# B&R Automation Studio project AAU12Segmenter (part 5)

#### linkMovement.st
```iecst
ACTION linkMovementProgram:
	//Setup
	positionContainerLinkMovement[0].Shuttle1.xPos := 0.120;
	positionContainerLinkMovement[0].Shuttle1.yPos := 0.120;
	positionContainerLinkMovement[0].Shuttle2.xPos := 0.360;
	positionContainerLinkMovement[0].Shuttle2.yPos := 0.360;
	positionContainerLinkMovement[0].Shuttle3.xPos := 0.360;
	positionContainerLinkMovement[0].Shuttle3.yPos := 0.120;
	positionContainerLinkMovement[0].Shuttle4.xPos := 0.120;
	positionContainerLinkMovement[0].Shuttle4.yPos := 0.360;

	positionContainerLinkMovement[1].Shuttle1.xPos := 0.060;
	positionContainerLinkMovement[1].Shuttle1.yPos := 0.060;
	positionContainerLinkMovement[1].Shuttle2.xPos := 0.180;
	positionContainerLinkMovement[1].Shuttle2.yPos := 0.180;
	positionContainerLinkMovement[1].Shuttle3.xPos := 0.180;
	positionContainerLinkMovement[1].Shuttle3.yPos := 0.060;
	positionContainerLinkMovement[1].Shuttle4.xPos := 0.060;
	positionContainerLinkMovement[1].Shuttle4.yPos := 0.180;

	positionContainerLinkMovement[2].Shuttle1.xPos := 0.120;
	positionContainerLinkMovement[2].Shuttle1.yPos := 0.120;
	positionContainerLinkMovement[2].Shuttle2.xPos := 0.360;
	positionContainerLinkMovement[2].Shuttle2.yPos := 0.360;
	positionContainerLinkMovement[2].Shuttle3.xPos := 0.360;
	positionContainerLinkMovement[2].Shuttle3.yPos := 0.120;
	positionContainerLinkMovement[2].Shuttle4.xPos := 0.120;
	positionContainerLinkMovement[2].Shuttle4.yPos := 0.360;

	positionContainerLinkMovement[3].Shuttle1.xPos := 0.300;
	positionContainerLinkMovement[3].Shuttle1.yPos := 0.060;
	positionContainerLinkMovement[3].Shuttle2.xPos := 0.420;
	positionContainerLinkMovement[3].Shuttle2.yPos := 0.180;
	positionContainerLinkMovement[3].Shuttle3.xPos := 0.420;
	positionContainerLinkMovement[3].Shuttle3.yPos := 0.060;
	positionContainerLinkMovement[3].Shuttle4.xPos := 0.300;
	positionContainerLinkMovement[3].Shuttle4.yPos := 0.180;

	positionContainerLinkMovement[4].Shuttle1.xPos := 0.120;
	positionContainerLinkMovement[4].Shuttle1.yPos := 0.120;
	positionContainerLinkMovement[4].Shuttle2.xPos := 0.360;
	positionContainerLinkMovement[4].Shuttle2.yPos := 0.360;
	positionContainerLinkMovement[4].Shuttle3.xPos := 0.360;
	positionContainerLinkMovement[4].Shuttle3.yPos := 0.120;
	positionContainerLinkMovement[4].Shuttle4.xPos := 0.120;
	positionContainerLinkMovement[4].Shuttle4.yPos := 0.360;

	positionContainerLinkMovement[5].Shuttle1.xPos := 0.300;
	positionContainerLinkMovement[5].Shuttle1.yPos := 0.300;
	positionContainerLinkMovement[5].Shuttle2.xPos := 0.420;
	positionContainerLinkMovement[5].Shuttle2.yPos := 0.420;
	positionContainerLinkMovement[5].Shuttle3.xPos := 0.420;
	positionContainerLinkMovement[5].Shuttle3.yPos := 0.300;
	positionContainerLinkMovement[5].Shuttle4.xPos := 0.300;
	positionContainerLinkMovement[5].Shuttle4.yPos := 0.420;

	positionContainerLinkMovement[6].Shuttle1.xPos := 0.120;
	positionContainerLinkMovement[6].Shuttle1.yPos := 0.120;
	positionContainerLinkMovement[6].Shuttle2.xPos := 0.360;
	positionContainerLinkMovement[6].Shuttle2.yPos := 0.360;
	positionContainerLinkMovement[6].Shuttle3.xPos := 0.360;
	positionContainerLinkMovement[6].Shuttle3.yPos := 0.120;
	positionContainerLinkMovement[6].Shuttle4.xPos := 0.120;
	positionContainerLinkMovement[6].Shuttle4.yPos := 0.360;

	positionContainerLinkMovementNew[0].initXPos := 0.540;
	positionContainerLinkMovementNew[0].initYPos := 0.300;
	positionContainerLinkMovementNew[1].initXPos := 0.540;
	positionContainerLinkMovementNew[1].initYPos := 0.420;
	positionContainerLinkMovementNew[2].initXPos := 0.660;
	positionContainerLinkMovementNew[2].initYPos := 0.540;
	positionContainerLinkMovementNew[3].initXPos := 0.660;
	positionContainerLinkMovementNew[3].initYPos := 0.660;

	positionContainerLinkMovementNew[4].initXPos := 0.120;
	positionContainerLinkMovementNew[4].initYPos := 0.120;
	positionContainerLinkMovementNew[5].initXPos := 0.120;
	positionContainerLinkMovementNew[5].initYPos := 0.240;
	positionContainerLinkMovementNew[6].initXPos := 0.240;
	positionContainerLinkMovementNew[6].initYPos := 0.240;
	positionContainerLinkMovementNew[7].initXPos := 0.240;
	positionContainerLinkMovementNew[7].initYPos := 0.120;
	positionContainerLinkMovementNew[8].initXPos := 0.540;
	positionContainerLinkMovementNew[8].initYPos := 0.900;
	positionContainerLinkMovementNew[9].initXPos := 0.660;
	positionContainerLinkMovementNew[9].initYPos := 0.900;

	CASE em.substate OF
		3000:
			em.description := 'Move all shuttles to prePos';
			em.cmd.sc := FALSE;
			tempShuttleCounter := 0;
			tempCounter := 0;
			em.substate := 3005;

		3005:
			em.description := 'Move shuttle to pre pos';
			tempShuttleCounter := 0;
			em.cmd.sc := FALSE;
			MC_BR_MoveInPlaneAsync_Acp6D_0.Parameters.Acceleration := gAcp6DCtrl.Par.Acceleration;
			MC_BR_MoveInPlaneAsync_Acp6D_0.Parameters.Velocity := gAcp6DCtrl.Par.Velocity;
			FOR i := 0 TO UINT_TO_USINT(localCurrentNumShuttles-1) DO
				MC_BR_MoveInPlaneAsync_Acp6D_0.Parameters.AsyncPar[i].Shuttle := ADR(gAcp6DCtrl.Status.ShuttleInfo[i].shuttleRef);
				MC_BR_MoveInPlaneAsync_Acp6D_0.Parameters.AsyncPar[i].X := positionContainerLinkMovementNew[i].initXPos;
				MC_BR_MoveInPlaneAsync_Acp6D_0.Parameters.AsyncPar[i].Y := positionContainerLinkMovementNew[i].initYPos;
			END_FOR
			MC_BR_MoveInPlaneAsync_Acp6D_0.Execute := TRUE;
			IF MC_BR_MoveInPlaneAsync_Acp6D_0.Done THEN
				MC_BR_MoveInPlaneAsync_Acp6D_0.Execute := FALSE;
				em.substate := 3010;
			END_IF

		3010:
			em.description := 'Move all shuttles to prePos';
			em.cmd.sc := FALSE;
			IF tempShuttleCounter > 3 THEN
				tempShuttleCounter := 0;
				em.substate := 3030;
			ELSE
				MC_BR_MoveInPlane_Acp6D_0.Parameters.Acceleration := gAcp6DCtrl.Par.Acceleration;
				MC_BR_MoveInPlane_Acp6D_0.Parameters.Velocity := gAcp6DCtrl.Par.Velocity;
				MC_BR_MoveInPlane_Acp6D_0.Parameters.Mode := 0; //Abs
				MC_BR_MoveInPlane_Acp6D_0.Shuttle := ADR(gAcp6DCtrl.Status.ShuttleInfo[tempShuttleCounter].shuttleRef);
				CASE tempShuttleCounter OF
					0:
						MC_BR_MoveInPlane_Acp6D_0.Parameters.Position.X := 0.540;
						MC_BR_MoveInPlane_Acp6D_0.Parameters.Position.Y := 0.300;
					1:
						MC_BR_MoveInPlane_Acp6D_0.Parameters.Position.X := 0.540;
						MC_BR_MoveInPlane_Acp6D_0.Parameters.Position.Y := 0.420;
					2:
						MC_BR_MoveInPlane_Acp6D_0.Parameters.Position.X := 0.660;
						MC_BR_MoveInPlane_Acp6D_0.Parameters.Position.Y := 0.540;
					3:
						MC_BR_MoveInPlane_Acp6D_0.Parameters.Position.X := 0.660;
						MC_BR_MoveInPlane_Acp6D_0.Parameters.Position.Y := 0.660;
				END_CASE

				MC_BR_MoveInPlane_Acp6D_0.Execute := TRUE;
				IF MC_BR_MoveInPlane_Acp6D_0.Acknowledge THEN
					MC_BR_MoveInPlane_Acp6D_0.Execute := FALSE;
					tempShuttleCounter := tempShuttleCounter + 1;
					em.substate := 3012;
				END_IF
			END_IF

		3012:
			em.description := 'Couple ShuttleGroup4_5_6_7';
			em.cmd.sc := FALSE;
			MC_BR_ShGroupCoupleCtrl_Acp6D_0.ShuttleGroup := shGroupShuttle5_6_7_8;
			MC_BR_ShGroupCoupleCtrl_Acp6D_0.Parameters.Option := 1; //Couple
			MC_BR_ShGroupCoupleCtrl_Acp6D_0.Execute := TRUE;
			IF MC_BR_ShGroupCoupleCtrl_Acp6D_0.Done THEN
				MC_BR_ShGroupCoupleCtrl_Acp6D_0.Execute := FALSE;
				em.substate := 3015;
			ELSIF MC_BR_ShGroupCoupleCtrl_Acp6D_0.Error THEN
				em.cmd.abort := TRUE;
			END_IF

		3015:
			em.description := 'DummyScan';
			em.cmd.sc := FALSE;
			em.substate := 3016;

		3016:
			em.cmd.sc := FALSE;
			MC_BR_MoveArc_Acp6D_0.Shuttle := ADR(gAcp6DCtrl.Status.ShuttleInfo[4].shuttleRef);
			MC_BR_MoveArc_Acp6D_0.Parameters.Mode := 0;
			MC_BR_MoveArc_Acp6D_0.Parameters.Option := mcACP6D_ARC_ANGULAR;
			MC_BR_MoveArc_Acp6D_0.Parameters.Direction := mcACP6D_ARC_CLOCKWISE;
			MC_BR_MoveArc_Acp6D_0.Parameters.Acceleration := 0.1;
			MC_BR_MoveArc_Acp6D_0.Parameters.Velocity := 0.5;
			MC_BR_MoveArc_Acp6D_0.Parameters.Angular.Angle := 628.318531;
			MC_BR_MoveArc_Acp6D_0.Parameters.Angular.Center.X := 0.180;
			MC_BR_MoveArc_Acp6D_0.Parameters.Angular.Center.Y := 0.180;
			MC_BR_MoveArc_Acp6D_0.Execute := TRUE;
			IF MC_BR_MoveArc_Acp6D_0.Acknowledge THEN
				MC_BR_MoveArc_Acp6D_0.Execute := FALSE;
				em.substate := 3020;
			END_IF

		3020:
			em.cmd.sc := FALSE;
			em.description := 'DummyScan';
			em.substate := 3010;

		3030:
			em.cmd.sc := FALSE;
			em.description := 'check shuttle state idle';
			IF gAcp6DCtrl.Status.ShuttleInfo[0].State = mcACP6D_SH_STATE_IDLING AND gAcp6DCtrl.Status.ShuttleInfo[1].State = mcACP6D_SH_STATE_IDLING
				AND gAcp6DCtrl.Status.ShuttleInfo[2].State = mcACP6D_SH_STATE_IDLING AND gAcp6DCtrl.Status.ShuttleInfo[3].State = mcACP6D_SH_STATE_IDLING AND MC_BR_AsmReadStatus_Acp6D_0.AssemblyReady THEN
				em.substate := 3035;
			END_IF

		3035:
			em.description := 'Couple ShuttleGroup1_2';
			em.cmd.sc := FALSE;
			MC_BR_ShGroupCoupleCtrl_Acp6D_0.ShuttleGroup := shGroupShuttle1_2;
			MC_BR_ShGroupCoupleCtrl_Acp6D_0.Parameters.Option := 1; //Couple
			MC_BR_ShGroupCoupleCtrl_Acp6D_0.Execute := TRUE;
			IF MC_BR_ShGroupCoupleCtrl_Acp6D_0.Done THEN
				MC_BR_ShGroupCoupleCtrl_Acp6D_0.Execute := FALSE;
				em.substate := 3040;
			ELSIF MC_BR_ShGroupCoupleCtrl_Acp6D_0.Error THEN
				em.cmd.abort := TRUE;
			END_IF

		3040:
			em.description := 'Couple ShuttleGroup1_2';
			em.cmd.sc := FALSE;
			MC_BR_ShGroupCoupleCtrl_Acp6D_0.ShuttleGroup := shGroupShuttle3_4;
			MC_BR_ShGroupCoupleCtrl_Acp6D_0.Parameters.Option := 1; //Couple
			MC_BR_ShGroupCoupleCtrl_Acp6D_0.Execute := TRUE;
			IF MC_BR_ShGroupCoupleCtrl_Acp6D_0.Done THEN
				MC_BR_ShGroupCoupleCtrl_Acp6D_0.Execute := FALSE;
				em.substate := 3050;
			ELSIF MC_BR_ShGroupCoupleCtrl_Acp6D_0.Error THEN
				em.cmd.abort := TRUE;
			END_IF

		3050:
			em.description := 'Move group 10 of shuttle around';
			em.cmd.sc := FALSE;
			IF tempCounter >= 3 THEN
				tempCounter := 0;
				em.substate := 3070;
			ELSE
				MC_BR_MoveInPlane_Acp6D_0.Shuttle := ADR(gAcp6DCtrl.Status.ShuttleInfo[0].shuttleRef);
				MC_BR_MoveInPlane_Acp6D_0.Parameters.Position.X := 0.660;
				MC_BR_MoveInPlane_Acp6D_0.Parameters.Position.Y := 0.540;
				MC_BR_MoveInPlane_Acp6D_0.Parameters.Path := 1; //X then Y
				MC_BR_MoveInPlane_Acp6D_0.Execute := TRUE;
				IF MC_BR_MoveInPlane_Acp6D_0.Acknowledge THEN
					MC_BR_MoveInPlane_Acp6D_0.Execute := FALSE;
					em.substate := 3060;
				END_IF
			END_IF

		3060:
			em.description := 'Move group of shuttle around';
			em.cmd.sc := FALSE;
			MC_BR_MoveInPlane_Acp6D_0.Shuttle := ADR(gAcp6DCtrl.Status.ShuttleInfo[0].shuttleRef);
			MC_BR_MoveInPlane_Acp6D_0.Parameters.Position.X := 0.540;
			MC_BR_MoveInPlane_Acp6D_0.Parameters.Position.Y := 0.300;
			MC_BR_MoveInPlane_Acp6D_0.Parameters.Velocity := gAcp6DCtrl.Par.Velocity;
			MC_BR_MoveInPlane_Acp6D_0.Parameters.Acceleration := gAcp6DCtrl.Par.Acceleration;
			MC_BR_MoveInPlane_Acp6D_0.Parameters.Path := 1; //X then Y
			MC_BR_MoveInPlane_Acp6D_0.Execute := TRUE;
			IF MC_BR_MoveInPlane_Acp6D_0.Acknowledge THEN
				MC_BR_MoveInPlane_Acp6D_0.Execute := FALSE;
				tempCounter := tempCounter + 1;
				em.substate := 3050;
			END_IF

		3070:
			em.description := 'Move group 11 of shuttle around';
			em.cmd.sc := FALSE;
			IF tempCounter >= 3 THEN
				tempCounter := 0;
				em.substate := 3090;
			ELSE
				MC_BR_MoveInPlane_Acp6D_0.Shuttle := ADR(gAcp6DCtrl.Status.ShuttleInfo[2].shuttleRef);
				MC_BR_MoveInPlane_Acp6D_0.Parameters.Position.X := 0.540;
				MC_BR_MoveInPlane_Acp6D_0.Parameters.Position.Y := 0.300;
				MC_BR_MoveInPlane_Acp6D_0.Parameters.Path := 1; //X then Y
				MC_BR_MoveInPlane_Acp6D_0.Execute := TRUE;
				IF MC_BR_MoveInPlane_Acp6D_0.Acknowledge THEN
					MC_BR_MoveInPlane_Acp6D_0.Execute := FALSE;
					em.substate := 3080;
				END_IF
			END_IF

		3080:
			em.description := 'Move group of shuttle around';
			em.cmd.sc := FALSE;
			MC_BR_MoveInPlane_Acp6D_0.Shuttle := ADR(gAcp6DCtrl.Status.ShuttleInfo[2].shuttleRef);
			MC_BR_MoveInPlane_Acp6D_0.Parameters.Position.X := 0.660;
			MC_BR_MoveInPlane_Acp6D_0.Parameters.Position.Y := 0.540;
			MC_BR_MoveInPlane_Acp6D_0.Parameters.Velocity := gAcp6DCtrl.Par.Velocity;
			MC_BR_MoveInPlane_Acp6D_0.Parameters.Acceleration := gAcp6DCtrl.Par.Acceleration;
			MC_BR_MoveInPlane_Acp6D_0.Parameters.Path := 1; //X then Y
			MC_BR_MoveInPlane_Acp6D_0.Execute := TRUE;
			IF MC_BR_MoveInPlane_Acp6D_0.Acknowledge THEN
				MC_BR_MoveInPlane_Acp6D_0.Execute := FALSE;
				tempCounter := tempCounter + 1;
				em.substate := 3070;
			END_IF

		3090:
			em.description := 'DeCouple ShuttleGroup1_2';
			em.cmd.sc := FALSE;
			MC_BR_ShGroupCoupleCtrl_Acp6D_0.ShuttleGroup := shGroupShuttle1_2;
			MC_BR_ShGroupCoupleCtrl_Acp6D_0.Parameters.Option := 0; //DeCouple
			MC_BR_ShGroupCoupleCtrl_Acp6D_0.Execute := TRUE;
			IF MC_BR_ShGroupCoupleCtrl_Acp6D_0.Done THEN
				MC_BR_ShGroupCoupleCtrl_Acp6D_0.Execute := FALSE;
				em.substate := 3100;
			ELSIF MC_BR_ShGroupCoupleCtrl_Acp6D_0.Error THEN
				em.cmd.abort := TRUE;
			END_IF

		3100:
			em.description := 'Wait for shuttle to reach pos';
			em.cmd.sc := FALSE;
			IF((gAcp6DCtrl.Status.ShuttleInfo[2].Position.X > 0.660 - MARGIN AND gAcp6DCtrl.Status.ShuttleInfo[2].Position.X < 0.660 + MARGIN) AND
				gAcp6DCtrl.Status.ShuttleInfo[2].Position.Y > 0.540 - MARGIN AND gAcp6DCtrl.Status.ShuttleInfo[2].Position.Y < 0.540 + MARGIN) THEN
				IF gAcp6DCtrl.Status.ShuttleInfo[2].State = mcACP6D_SH_STATE_IDLING THEN
					em.substate := 3110;
				END_IF
			END_IF

		3110:
			em.description := 'Move right group up';
			em.cmd.sc := FALSE;
			MC_BR_MoveInPlane_Acp6D_0.Shuttle := ADR(gAcp6DCtrl.Status.ShuttleInfo[2].shuttleRef);
			MC_BR_MoveInPlane_Acp6D_0.Parameters.Position.X := 0.540;
			MC_BR_MoveInPlane_Acp6D_0.Parameters.Position.Y := 0.540;
			MC_BR_MoveInPlane_Acp6D_0.Parameters.Velocity := gAcp6DCtrl.Par.Velocity;
			MC_BR_MoveInPlane_Acp6D_0.Parameters.Acceleration := gAcp6DCtrl.Par.Acceleration;
			MC_BR_MoveInPlane_Acp6D_0.Parameters.Path := 0; //Direct
			MC_BR_MoveInPlane_Acp6D_0.Execute := TRUE;
			IF MC_BR_MoveInPlane_Acp6D_0.Acknowledge THEN
				MC_BR_MoveInPlane_Acp6D_0.Execute := FALSE;
				em.substate := 3120;
			END_IF

		3120:
			em.description := 'Couple ShuttleGroup1_2';
			em.cmd.sc := FALSE;
			MC_BR_ShGroupCoupleCtrl_Acp6D_0.ShuttleGroup := shGroupShuttle3_4;
			MC_BR_ShGroupCoupleCtrl_Acp6D_0.Parameters.Option := 0; //DeCouple
			MC_BR_ShGroupCoupleCtrl_Acp6D_0.Execute := TRUE;
			IF MC_BR_ShGroupCoupleCtrl_Acp6D_0.Done THEN
				MC_BR_ShGroupCoupleCtrl_Acp6D_0.Execute := FALSE;
				em.substate := 3130;
			ELSIF MC_BR_ShGroupCoupleCtrl_Acp6D_0.Error THEN
				em.cmd.abort := TRUE;
			END_IF

		3130:
			em.description := 'rotationMove part 1';
			em.cmd.sc := FALSE;
			MC_BR_MoveInPlane_Acp6D_0.Shuttle := ADR(gAcp6DCtrl.Status.ShuttleInfo[1].shuttleRef);
			MC_BR_MoveInPlane_Acp6D_0.Parameters.Position.X := 0.660;
			MC_BR_MoveInPlane_Acp6D_0.Parameters.Position.Y := 0.300;
			MC_BR_MoveInPlane_Acp6D_0.Parameters.Velocity := gAcp6DCtrl.Par.Velocity;
			MC_BR_MoveInPlane_Acp6D_0.Parameters.Acceleration := gAcp6DCtrl.Par.Acceleration;
			MC_BR_MoveInPlane_Acp6D_0.Parameters.Path := 1; //X then Y
			MC_BR_MoveInPlane_Acp6D_0.Execute := TRUE;
			IF MC_BR_MoveInPlane_Acp6D_0.Acknowledge THEN
				MC_BR_MoveInPlane_Acp6D_0.Execute := FALSE;
				em.substate := 3140;
			END_IF

		3140:
			em.description := 'rotationMove part 2';
			em.cmd.sc := FALSE;
			MC_BR_MoveInPlane_Acp6D_0.Shuttle := ADR(gAcp6DCtrl.Status.ShuttleInfo[3].shuttleRef);
			MC_BR_MoveInPlane_Acp6D_0.Parameters.Position.X := 0.660;
			MC_BR_MoveInPlane_Acp6D_0.Parameters.Position.Y := 0.420;
			MC_BR_MoveInPlane_Acp6D_0.Parameters.Velocity := gAcp6DCtrl.Par.Velocity;
			MC_BR_MoveInPlane_Acp6D_0.Parameters.Acceleration := gAcp6DCtrl.Par.Acceleration;
			MC_BR_MoveInPlane_Acp6D_0.Parameters.Path := 1; //X then Y
			MC_BR_MoveInPlane_Acp6D_0.Execute := TRUE;
			IF MC_BR_MoveInPlane_Acp6D_0.Acknowledge THEN
				MC_BR_MoveInPlane_Acp6D_0.Execute := FALSE;
				em.substate := 3150;
			END_IF

		3150:
			em.description := 'rotationMove part 3';
			em.cmd.sc := FALSE;
			MC_BR_MoveInPlane_Acp6D_0.Shuttle := ADR(gAcp6DCtrl.Status.ShuttleInfo[3].shuttleRef);
			MC_BR_MoveInPlane_Acp6D_0.Parameters.Position.X := 0.540;
			MC_BR_MoveInPlane_Acp6D_0.Parameters.Velocity := gAcp6DCtrl.Par.Velocity;
			MC_BR_MoveInPlane_Acp6D_0.Parameters.Acceleration := gAcp6DCtrl.Par.Acceleration;
			MC_BR_MoveInPlane_Acp6D_0.Parameters.Position.Y := 0.420;
			MC_BR_MoveInPlane_Acp6D_0.Parameters.Path := 0; //direct
			MC_BR_MoveInPlane_Acp6D_0.Execute := TRUE;
			IF MC_BR_MoveInPlane_Acp6D_0.Acknowledge THEN
				MC_BR_MoveInPlane_Acp6D_0.Execute := FALSE;
				em.substate := 3160;
			END_IF

		3160:
			em.description := 'Check switch is done part 1';
			em.cmd.sc := FALSE;
			IF((gAcp6DCtrl.Status.ShuttleInfo[3].Position.X > 0.540 - MARGIN AND gAcp6DCtrl.Status.ShuttleInfo[3].Position.X < 0.540 + MARGIN) AND
				gAcp6DCtrl.Status.ShuttleInfo[3].Position.Y > 0.420 - MARGIN AND gAcp6DCtrl.Status.ShuttleInfo[3].Position.Y < 0.420 + MARGIN) THEN
				IF gAcp6DCtrl.Status.ShuttleInfo[3].State = mcACP6D_SH_STATE_IDLING THEN
					em.substate := 3170;
				END_IF
			END_IF

		3170:
			em.description := 'rotationMove part 4';
			em.cmd.sc := FALSE;
			MC_BR_MoveInPlane_Acp6D_0.Shuttle := ADR(gAcp6DCtrl.Status.ShuttleInfo[1].shuttleRef);
			MC_BR_MoveInPlane_Acp6D_0.Parameters.Position.X := 0.540;
			MC_BR_MoveInPlane_Acp6D_0.Parameters.Position.Y := 0.660;
			MC_BR_MoveInPlane_Acp6D_0.Parameters.Velocity := gAcp6DCtrl.Par.Velocity;
			MC_BR_MoveInPlane_Acp6D_0.Parameters.Acceleration := gAcp6DCtrl.Par.Acceleration;
			MC_BR_MoveInPlane_Acp6D_0.Parameters.Path := 2; //Y then X
			MC_BR_MoveInPlane_Acp6D_0.Execute := TRUE;
			IF MC_BR_MoveInPlane_Acp6D_0.Acknowledge THEN
				MC_BR_MoveInPlane_Acp6D_0.Execute := FALSE;
				em.substate := 3180;
			END_IF

		3180:
			em.description := 'Check switch is done part 2';
			em.cmd.sc := FALSE;
			IF((gAcp6DCtrl.Status.ShuttleInfo[1].Position.X > 0.540 - MARGIN AND gAcp6DCtrl.Status.ShuttleInfo[1].Position.X < 0.540 + MARGIN) AND
				gAcp6DCtrl.Status.ShuttleInfo[1].Position.Y > 0.660 - MARGIN AND gAcp6DCtrl.Status.ShuttleInfo[1].Position.Y < 0.660 + MARGIN) THEN
				IF gAcp6DCtrl.Status.ShuttleInfo[1].State = mcACP6D_SH_STATE_IDLING THEN
					em.substate := 3190;
				END_IF
			END_IF

		3190:
			em.description := 'Couple ShuttleGroup1_4';
			em.cmd.sc := FALSE;
			MC_BR_ShGroupCoupleCtrl_Acp6D_0.ShuttleGroup := shGroupShuttle1_4;
			MC_BR_ShGroupCoupleCtrl_Acp6D_0.Parameters.Option := 1; //Couple
			MC_BR_ShGroupCoupleCtrl_Acp6D_0.Execute := TRUE;
			IF MC_BR_ShGroupCoupleCtrl_Acp6D_0.Done THEN
				MC_BR_ShGroupCoupleCtrl_Acp6D_0.Execute := FALSE;
				em.substate := 3200;
			ELSIF MC_BR_ShGroupCoupleCtrl_Acp6D_0.Error THEN
				em.cmd.abort := TRUE;
			END_IF

		3200:
			em.description := 'Couple ShuttleGroup2_3';
			em.cmd.sc := FALSE;
			MC_BR_ShGroupCoupleCtrl_Acp6D_0.ShuttleGroup := shGroupShuttle2_3;
			MC_BR_ShGroupCoupleCtrl_Acp6D_0.Parameters.Option := 1; //Couple
			MC_BR_ShGroupCoupleCtrl_Acp6D_0.Execute := TRUE;
			IF MC_BR_ShGroupCoupleCtrl_Acp6D_0.Done THEN
				MC_BR_ShGroupCoupleCtrl_Acp6D_0.Execute := FALSE;
				em.substate := 3210;
			ELSIF MC_BR_ShGroupCoupleCtrl_Acp6D_0.Error THEN
				em.cmd.abort := TRUE;
			END_IF

		3210:
			em.description := 'Move right side down';
			em.cmd.sc := FALSE;
			MC_BR_MoveInPlane_Acp6D_0.Shuttle := ADR(gAcp6DCtrl.Status.ShuttleInfo[2].shuttleRef);
			MC_BR_MoveInPlane_Acp6D_0.Parameters.Position.X := 0.660;
			MC_BR_MoveInPlane_Acp6D_0.Parameters.Position.Y := 0.540;
			MC_BR_MoveInPlane_Acp6D_0.Parameters.Velocity := gAcp6DCtrl.Par.Velocity;
			MC_BR_MoveInPlane_Acp6D_0.Parameters.Acceleration := gAcp6DCtrl.Par.Acceleration;
			MC_BR_MoveInPlane_Acp6D_0.Parameters.Path := 0; //direct
			MC_BR_MoveInPlane_Acp6D_0.Execute := TRUE;
			IF MC_BR_MoveInPlane_Acp6D_0.Acknowledge THEN
				MC_BR_MoveInPlane_Acp6D_0.Execute := FALSE;
				em.substate := 3230;
			END_IF

		3230:
			em.description := 'Move group 12 of shuttle around';
			em.cmd.sc := FALSE;
			IF tempCounter >= 3 THEN
				tempCounter := 0;
				em.substate := 3250;
			ELSE
				MC_BR_MoveInPlane_Acp6D_0.Shuttle := ADR(gAcp6DCtrl.Status.ShuttleInfo[0].shuttleRef);
				MC_BR_MoveInPlane_Acp6D_0.Parameters.Position.X := 0.660;
				MC_BR_MoveInPlane_Acp6D_0.Parameters.Position.Y := 0.540;
				MC_BR_MoveInPlane_Acp6D_0.Parameters.Path := 2; //Y then X
				MC_BR_MoveInPlane_Acp6D_0.Execute := TRUE;
				IF MC_BR_MoveInPlane_Acp6D_0.Acknowledge THEN
					MC_BR_MoveInPlane_Acp6D_0.Execute := FALSE;
					em.substate := 3240;
				END_IF
			END_IF

		3240:
			em.description := 'Move group of shuttle around';
			em.cmd.sc := FALSE;
			MC_BR_MoveInPlane_Acp6D_0.Shuttle := ADR(gAcp6DCtrl.Status.ShuttleInfo[0].shuttleRef);
			MC_BR_MoveInPlane_Acp6D_0.Parameters.Position.X := 0.540;
			MC_BR_MoveInPlane_Acp6D_0.Parameters.Position.Y := 0.300;
			MC_BR_MoveInPlane_Acp6D_0.Parameters.Velocity := gAcp6DCtrl.Par.Velocity;
			MC_BR_MoveInPlane_Acp6D_0.Parameters.Acceleration := gAcp6DCtrl.Par.Acceleration;
			MC_BR_MoveInPlane_Acp6D_0.Parameters.Path := 2; //Y then X
			MC_BR_MoveInPlane_Acp6D_0.Execute := TRUE;
			IF MC_BR_MoveInPlane_Acp6D_0.Acknowledge THEN
				MC_BR_MoveInPlane_Acp6D_0.Execute := FALSE;
				tempCounter := tempCounter + 1;
				em.substate := 3230;
			END_IF

		3250:
			em.description := 'Move group 13 of shuttle around';
			em.cmd.sc := FALSE;
			IF tempCounter >= 3 THEN
				tempCounter := 0;
				em.substate := 3270;
			ELSE
				MC_BR_MoveInPlane_Acp6D_0.Shuttle := ADR(gAcp6DCtrl.Status.ShuttleInfo[2].shuttleRef);
				MC_BR_MoveInPlane_Acp6D_0.Parameters.Position.X := 0.540;
				MC_BR_MoveInPlane_Acp6D_0.Parameters.Position.Y := 0.300;
				MC_BR_MoveInPlane_Acp6D_0.Parameters.Path := 2; //Y then X
				MC_BR_MoveInPlane_Acp6D_0.Execute := TRUE;
				IF MC_BR_MoveInPlane_Acp6D_0.Acknowledge THEN
					MC_BR_MoveInPlane_Acp6D_0.Execute := FALSE;
					em.substate := 3260;
				END_IF
			END_IF

		3260:
			em.description := 'Move group of shuttle around';
			em.cmd.sc := FALSE;
			MC_BR_MoveInPlane_Acp6D_0.Shuttle := ADR(gAcp6DCtrl.Status.ShuttleInfo[2].shuttleRef);
			MC_BR_MoveInPlane_Acp6D_0.Parameters.Position.X := 0.660;
			MC_BR_MoveInPlane_Acp6D_0.Parameters.Position.Y := 0.540;
			MC_BR_MoveInPlane_Acp6D_0.Parameters.Velocity := gAcp6DCtrl.Par.Velocity;
			MC_BR_MoveInPlane_Acp6D_0.Parameters.Acceleration := gAcp6DCtrl.Par.Acceleration;
			MC_BR_MoveInPlane_Acp6D_0.Parameters.Path := 2; //Y then X
			MC_BR_MoveInPlane_Acp6D_0.Execute := TRUE;
			IF MC_BR_MoveInPlane_Acp6D_0.Acknowledge THEN
				MC_BR_MoveInPlane_Acp6D_0.Execute := FALSE;
				tempCounter := tempCounter + 1;
				em.substate := 3250;
			END_IF

		3270:
			em.cmd.sc := FALSE;
			IF((gAcp6DCtrl.Status.ShuttleInfo[2].Position.X > 0.660 - MARGIN AND gAcp6DCtrl.Status.ShuttleInfo[2].Position.X < 0.660 + MARGIN) AND
				gAcp6DCtrl.Status.ShuttleInfo[2].Position.Y > 0.540 - MARGIN AND gAcp6DCtrl.Status.ShuttleInfo[2].Position.Y < 0.540 + MARGIN) THEN
				IF gAcp6DCtrl.Status.ShuttleInfo[2].State = mcACP6D_SH_STATE_IDLING THEN
					em.substate := 3280;
				END_IF
			END_IF

		3280:
			em.description := 'Move right group up';
			em.cmd.sc := FALSE;
			MC_BR_MoveInPlane_Acp6D_0.Shuttle := ADR(gAcp6DCtrl.Status.ShuttleInfo[2].shuttleRef);
			MC_BR_MoveInPlane_Acp6D_0.Parameters.Position.X := 0.540;
			MC_BR_MoveInPlane_Acp6D_0.Parameters.Position.Y := 0.540;
			MC_BR_MoveInPlane_Acp6D_0.Parameters.Velocity := gAcp6DCtrl.Par.Velocity;
			MC_BR_MoveInPlane_Acp6D_0.Parameters.Acceleration := gAcp6DCtrl.Par.Acceleration;
			MC_BR_MoveInPlane_Acp6D_0.Parameters.Path := 0; //Direct
			MC_BR_MoveInPlane_Acp6D_0.Execute := TRUE;
			IF MC_BR_MoveInPlane_Acp6D_0.Acknowledge THEN
				MC_BR_MoveInPlane_Acp6D_0.Execute := FALSE;
				em.substate := 3290;
			END_IF

		3290:
			em.description := 'DeCouple ShuttleGroup1_4';
			em.cmd.sc := FALSE;
			MC_BR_ShGroupCoupleCtrl_Acp6D_0.ShuttleGroup := shGroupShuttle1_4;
			MC_BR_ShGroupCoupleCtrl_Acp6D_0.Parameters.Option := 0; //DeCouple
			MC_BR_ShGroupCoupleCtrl_Acp6D_0.Execute := TRUE;
			IF MC_BR_ShGroupCoupleCtrl_Acp6D_0.Done THEN
				MC_BR_ShGroupCoupleCtrl_Acp6D_0.Execute := FALSE;
				em.substate := 3300;
			ELSIF MC_BR_ShGroupCoupleCtrl_Acp6D_0.Error THEN
				em.cmd.abort := TRUE;
			END_IF

		3300:
			em.description := 'DeCouple ShuttleGroup2_3';
			em.cmd.sc := FALSE;
			MC_BR_ShGroupCoupleCtrl_Acp6D_0.ShuttleGroup := shGroupShuttle2_3;
			MC_BR_ShGroupCoupleCtrl_Acp6D_0.Parameters.Option := 0; //DeCouple
			MC_BR_ShGroupCoupleCtrl_Acp6D_0.Execute := TRUE;
			IF MC_BR_ShGroupCoupleCtrl_Acp6D_0.Done THEN
				MC_BR_ShGroupCoupleCtrl_Acp6D_0.Execute := FALSE;
				em.substate := 3310;
			ELSIF MC_BR_ShGroupCoupleCtrl_Acp6D_0.Error THEN
				em.cmd.abort := TRUE;
			END_IF

		3310:
			em.description := 'rotationMove part 1';
			em.cmd.sc := FALSE;
			MC_BR_MoveInPlane_Acp6D_0.Shuttle := ADR(gAcp6DCtrl.Status.ShuttleInfo[3].shuttleRef);
			MC_BR_MoveInPlane_Acp6D_0.Parameters.Position.X := 0.660;
			MC_BR_MoveInPlane_Acp6D_0.Parameters.Position.Y := 0.300;
			MC_BR_MoveInPlane_Acp6D_0.Parameters.Velocity := gAcp6DCtrl.Par.Velocity;
			MC_BR_MoveInPlane_Acp6D_0.Parameters.Acceleration := gAcp6DCtrl.Par.Acceleration;
			MC_BR_MoveInPlane_Acp6D_0.Parameters.Path := 1; //X then Y
			MC_BR_MoveInPlane_Acp6D_0.Execute := TRUE;
			IF MC_BR_MoveInPlane_Acp6D_0.Acknowledge THEN
				MC_BR_MoveInPlane_Acp6D_0.Execute := FALSE;
				em.substate := 3320;
			END_IF

		3320:
			em.description := 'rotationMove part 2';
			em.cmd.sc := FALSE;
			MC_BR_MoveInPlane_Acp6D_0.Shuttle := ADR(gAcp6DCtrl.Status.ShuttleInfo[1].shuttleRef);
			MC_BR_MoveInPlane_Acp6D_0.Parameters.Position.X := 0.660;
			MC_BR_MoveInPlane_Acp6D_0.Parameters.Position.Y := 0.420;
			MC_BR_MoveInPlane_Acp6D_0.Parameters.Velocity := gAcp6DCtrl.Par.Velocity;
			MC_BR_MoveInPlane_Acp6D_0.Parameters.Acceleration := gAcp6DCtrl.Par.Acceleration;
			MC_BR_MoveInPlane_Acp6D_0.Parameters.Path := 1; //X then Y
			MC_BR_MoveInPlane_Acp6D_0.Execute := TRUE;
			IF MC_BR_MoveInPlane_Acp6D_0.Acknowledge THEN
				MC_BR_MoveInPlane_Acp6D_0.Execute := FALSE;
				em.substate := 3330;
			END_IF

		3330:
			em.description := 'rotationMove part 3';
			em.cmd.sc := FALSE;
			MC_BR_MoveInPlane_Acp6D_0.Shuttle := ADR(gAcp6DCtrl.Status.ShuttleInfo[1].shuttleRef);
			MC_BR_MoveInPlane_Acp6D_0.Parameters.Position.X := 0.540;
			MC_BR_MoveInPlane_Acp6D_0.Parameters.Position.Y := 0.420;
			MC_BR_MoveInPlane_Acp6D_0.Parameters.Velocity := gAcp6DCtrl.Par.Velocity;
			MC_BR_MoveInPlane_Acp6D_0.Parameters.Acceleration := gAcp6DCtrl.Par.Acceleration;
			MC_BR_MoveInPlane_Acp6D_0.Parameters.Path := 0; //direct
			MC_BR_MoveInPlane_Acp6D_0.Execute := TRUE;
			IF MC_BR_MoveInPlane_Acp6D_0.Acknowledge THEN
				MC_BR_MoveInPlane_Acp6D_0.Execute := FALSE;
				em.substate := 3340;
			END_IF

		3340:
			em.cmd.sc := FALSE;
			IF((gAcp6DCtrl.Status.ShuttleInfo[1].Position.X > 0.540 - MARGIN AND gAcp6DCtrl.Status.ShuttleInfo[1].Position.X < 0.540 + MARGIN) AND
				gAcp6DCtrl.Status.ShuttleInfo[1].Position.Y > 0.420 - MARGIN AND gAcp6DCtrl.Status.ShuttleInfo[1].Position.Y < 0.420 + MARGIN) THEN
				IF gAcp6DCtrl.Status.ShuttleInfo[1].State = mcACP6D_SH_STATE_IDLING THEN
					em.substate := 3350;
				END_IF
			END_IF

		3350:
			em.description := 'rotationMove part 4';
			em.cmd.sc := FALSE;
			MC_BR_MoveInPlane_Acp6D_0.Shuttle := ADR(gAcp6DCtrl.Status.ShuttleInfo[3].shuttleRef);
			MC_BR_MoveInPlane_Acp6D_0.Parameters.Position.X := 0.540;
			MC_BR_MoveInPlane_Acp6D_0.Parameters.Position.Y := 0.660;
			MC_BR_MoveInPlane_Acp6D_0.Parameters.Velocity := gAcp6DCtrl.Par.Velocity;
			MC_BR_MoveInPlane_Acp6D_0.Parameters.Acceleration := gAcp6DCtrl.Par.Acceleration;
			MC_BR_MoveInPlane_Acp6D_0.Parameters.Path := 2; //Y then X
			MC_BR_MoveInPlane_Acp6D_0.Execute := TRUE;
			IF MC_BR_MoveInPlane_Acp6D_0.Acknowledge THEN
				MC_BR_MoveInPlane_Acp6D_0.Execute := FALSE;
				em.substate := 3360;
			END_IF

		3360:
			em.cmd.sc := FALSE;
			IF((gAcp6DCtrl.Status.ShuttleInfo[3].Position.X > 0.540 - MARGIN AND gAcp6DCtrl.Status.ShuttleInfo[3].Position.X < 0.540 + MARGIN) AND
				gAcp6DCtrl.Status.ShuttleInfo[3].Position.Y > 0.660 - MARGIN AND gAcp6DCtrl.Status.ShuttleInfo[3].Position.Y < 0.660 + MARGIN) THEN
				IF gAcp6DCtrl.Status.ShuttleInfo[3].State = mcACP6D_SH_STATE_IDLING THEN
					em.substate := 3370;
				END_IF
			END_IF

		3370:
			//Check if next program is selected
			em.cmd.sc := FALSE;
			IF em.status.parent.state <> STATE_EXECUTE THEN
				em.substate := 3380;
			ELSE
				em.substate := 3030;
			END_IF

		3380:
			MC_BR_AsmStop_Acp6D_0.Execute := TRUE;
			em.cmd.sc := FALSE;
			IF MC_BR_AsmStop_Acp6D_0.Done THEN
				MC_BR_AsmStop_Acp6D_0.Execute := FALSE;
				em.substate := 3390;
			END_IF

		3390:
			em.description := 'Couple ShuttleGroup4_5_6_7';
			em.cmd.sc := FALSE;
			MC_BR_ShGroupCoupleCtrl_Acp6D_0.ShuttleGroup := shGroupShuttle5_6_7_8;
			MC_BR_ShGroupCoupleCtrl_Acp6D_0.Parameters.Option := 0; //DeCouple
			MC_BR_ShGroupCoupleCtrl_Acp6D_0.Execute := TRUE;
			IF MC_BR_ShGroupCoupleCtrl_Acp6D_0.Done THEN
				MC_BR_ShGroupCoupleCtrl_Acp6D_0.Execute := FALSE;
				em.substate := 3400;
				em.cmd.sc := TRUE;
			ELSIF MC_BR_ShGroupCoupleCtrl_Acp6D_0.Error THEN
				em.cmd.abort := TRUE;
			END_IF

		3400:
			em.cmd.sc := TRUE;

	END_CASE

	TON_0();

END_ACTION
```

#### conveyourStationMovement.st
```iecst
ACTION conveyorStationSetup:
	// Setup
	// Reset all workstations
	FOR i := 0 TO NR_OF_WORKSTATIONS DO
		gWorkstations[i].par.xLocation										:= 0.0;
		gWorkstations[i].par.yLocation										:= 0.0;
		gWorkstations[i].par.nextStationSelector							:= '0';
		gWorkstations[i].par.processTime									:= 0;
		gWorkstations[i].par.pathRouting									:= 0;
		gWorkstations[i].par.ArcMovement									:= FALSE;
		gWorkstations[i].par.landBeforeProcess								:= FALSE;
	END_FOR

	gWorkstations[0].par.xLocation										:= 0.180;
	gWorkstations[0].par.yLocation										:= 0.060;
	gWorkstations[0].par.nextStationSelector							:= '1';
	gWorkstations[0].par.processTime									:= 1;
	gWorkstations[0].par.pathRouting									:= 1;
	gWorkstations[0].par.ArcMovement									:= FALSE;
	gWorkstations[0].par.landBeforeProcess								:= FALSE;

	gWorkstations[1].par.xLocation										:= 0.660;
	gWorkstations[1].par.yLocation										:= 0.060;
	gWorkstations[1].par.nextStationSelector							:= '3';
	gWorkstations[1].par.processTime									:= 2;
	gWorkstations[1].par.pathRouting									:= 2;
	gWorkstations[1].par.ArcMovement									:= FALSE;
	gWorkstations[1].par.landBeforeProcess								:= FALSE;

	//Not in use
	gWorkstations[2].par.xLocation										:= 0.000;
	gWorkstations[2].par.yLocation										:= 0.000;
	gWorkstations[2].par.nextStationSelector							:= '0';
	gWorkstations[2].par.processTime									:= 0;
	gWorkstations[2].par.pathRouting									:= 2;
	gWorkstations[2].par.ArcMovement									:= FALSE;
	gWorkstations[2].par.landBeforeProcess								:= FALSE;

	gWorkstations[3].par.xLocation										:= 0.660;
	gWorkstations[3].par.yLocation										:= 0.300;
	gWorkstations[3].par.nextStationSelector							:= '4';
	gWorkstations[3].par.processTime									:= 1;
	gWorkstations[3].par.pathRouting									:= 2;
	gWorkstations[3].par.ArcMovement									:= FALSE;
	gWorkstations[3].par.landBeforeProcess								:= FALSE;

	gWorkstations[4].par.xLocation										:= 0.540;
	gWorkstations[4].par.yLocation										:= 0.900;
	gWorkstations[4].par.nextStationSelector							:= '5';
	gWorkstations[4].par.processTime									:= 1;
	gWorkstations[4].par.pathRouting									:= 2;
	gWorkstations[4].par.ArcMovement									:= FALSE;
	gWorkstations[4].par.landBeforeProcess								:= FALSE;

	gWorkstations[5].par.xLocation										:= 0.420;
	gWorkstations[5].par.yLocation										:= 0.420;
	gWorkstations[5].par.nextStationSelector							:= '6';
	gWorkstations[5].par.processTime									:= 2;
	gWorkstations[5].par.pathRouting									:= 0;
	gWorkstations[5].par.ArcMovement									:= FALSE;
	gWorkstations[5].par.landBeforeProcess								:= FALSE;

	gWorkstations[6].par.xLocation										:= 0.060;
	gWorkstations[6].par.yLocation										:= 0.420;
	gWorkstations[6].par.nextStationSelector							:= '0';
	gWorkstations[6].par.processTime									:= 1;
	gWorkstations[6].par.pathRouting									:= 2;
	gWorkstations[6].par.ArcMovement									:= FALSE;
	gWorkstations[6].par.landBeforeProcess								:= FALSE;

	gWorkstations[7].par.xLocation										:= 0.300;
	gWorkstations[7].par.yLocation										:= 0.900;
	gWorkstations[7].par.nextStationSelector							:= '6';
	gWorkstations[7].par.processTime									:= 2;
	gWorkstations[7].par.pathRouting									:= 2;
	gWorkstations[7].par.ArcMovement									:= FALSE;
	gWorkstations[7].par.landBeforeProcess								:= FALSE;

	positionContainerWorkstationMov[0].initXPos							:= 0.060;
	positionContainerWorkstationMov[0].initYPos							:= 0.060;
	positionContainerWorkstationMov[1].initXPos							:= 0.180;
	positionContainerWorkstationMov[1].initYPos							:= 0.060;
	positionContainerWorkstationMov[2].initXPos							:= 0.420;
	positionContainerWorkstationMov[2].initYPos							:= 0.060;
	positionContainerWorkstationMov[3].initXPos							:= 0.540;
	positionContainerWorkstationMov[3].initYPos							:= 0.300;

	positionContainerWorkstationMov[4].initXPos							:= 0.060;
	positionContainerWorkstationMov[4].initYPos							:= 0.180;
	positionContainerWorkstationMov[5].initXPos							:= 0.060;
	positionContainerWorkstationMov[5].initYPos							:= 0.300;
	positionContainerWorkstationMov[6].initXPos							:= 0.660;
	positionContainerWorkstationMov[6].initYPos							:= 0.300;
	positionContainerWorkstationMov[7].initXPos							:= 0.540;
	positionContainerWorkstationMov[7].initYPos							:= 0.900;

	CASE em.substate OF
		9000:
			em.description := 'Move shuttle to pre pos';
			tempShuttleCounter := 0;
			MC_BR_MoveInPlaneAsync_Acp6D_0.Parameters.Acceleration := gAcp6DCtrl.Par.Acceleration;
			MC_BR_MoveInPlaneAsync_Acp6D_0.Parameters.Velocity := gAcp6DCtrl.Par.Velocity;
			FOR i := 0 TO UINT_TO_USINT(localCurrentNumShuttles-1) DO
				MC_BR_MoveInPlaneAsync_Acp6D_0.Parameters.AsyncPar[i].Shuttle := ADR(gAcp6DCtrl.Status.ShuttleInfo[i].shuttleRef);
				MC_BR_MoveInPlaneAsync_Acp6D_0.Parameters.AsyncPar[i].X := positionContainerWorkstationMov[i].initXPos;
				MC_BR_MoveInPlaneAsync_Acp6D_0.Parameters.AsyncPar[i].Y := positionContainerWorkstationMov[i].initYPos;
			END_FOR
			MC_BR_MoveInPlaneAsync_Acp6D_0.Execute := TRUE;
			IF MC_BR_MoveInPlaneAsync_Acp6D_0.Acknowledge THEN
				MC_BR_MoveInPlaneAsync_Acp6D_0.Execute := FALSE;
				em.substate := 9001;
			END_IF

		9001:
			MC_BR_MoveInPlane_Acp6D_0.Parameters.Acceleration := gAcp6DCtrl.Par.Acceleration;
			MC_BR_MoveInPlane_Acp6D_0.Parameters.Velocity := gAcp6DCtrl.Par.Velocity;
			MC_BR_MoveInPlane_Acp6D_0.Shuttle := ADR(gAcp6DCtrl.Status.ShuttleInfo[0].shuttleRef);;
			MC_BR_MoveInPlane_Acp6D_0.Parameters.Position.X := gWorkstations[0].par.xLocation;;
			MC_BR_MoveInPlane_Acp6D_0.Parameters.Position.Y := gWorkstations[0].par.yLocation;
			MC_BR_MoveInPlane_Acp6D_0.Parameters.Path := 0; //Y then X
			MC_BR_MoveInPlane_Acp6D_0.Parameters.Mode := 0;
			MC_BR_MoveInPlane_Acp6D_0.Execute := TRUE;
			IF MC_BR_MoveInPlane_Acp6D_0.Acknowledge THEN
				MC_BR_MoveInPlane_Acp6D_0.Execute := FALSE;
				em.substate := 9002;
			END_IF

		9002:
			MC_BR_MoveInPlane_Acp6D_0.Parameters.Acceleration := gAcp6DCtrl.Par.Acceleration;
			MC_BR_MoveInPlane_Acp6D_0.Parameters.Velocity := gAcp6DCtrl.Par.Velocity;
			MC_BR_MoveInPlane_Acp6D_0.Shuttle := ADR(gAcp6DCtrl.Status.ShuttleInfo[2].shuttleRef);;
			MC_BR_MoveInPlane_Acp6D_0.Parameters.Position.X := gWorkstations[1].par.xLocation;;
			MC_BR_MoveInPlane_Acp6D_0.Parameters.Position.Y := gWorkstations[1].par.yLocation;
			MC_BR_MoveInPlane_Acp6D_0.Parameters.Path := 0; //Y then X
			MC_BR_MoveInPlane_Acp6D_0.Parameters.Mode := 0;
			MC_BR_MoveInPlane_Acp6D_0.Execute := TRUE;
			IF MC_BR_MoveInPlane_Acp6D_0.Acknowledge THEN
				MC_BR_MoveInPlane_Acp6D_0.Execute := FALSE;
				em.substate := 9003;
			END_IF

		9003:
			MC_BR_MoveInPlane_Acp6D_0.Parameters.Acceleration := gAcp6DCtrl.Par.Acceleration;
			MC_BR_MoveInPlane_Acp6D_0.Parameters.Velocity := gAcp6DCtrl.Par.Velocity;
			MC_BR_MoveInPlane_Acp6D_0.Shuttle := ADR(gAcp6DCtrl.Status.ShuttleInfo[3].shuttleRef);;
			MC_BR_MoveInPlane_Acp6D_0.Parameters.Position.X := gWorkstations[3].par.xLocation;;
			MC_BR_MoveInPlane_Acp6D_0.Parameters.Position.Y := gWorkstations[3].par.yLocation;
			MC_BR_MoveInPlane_Acp6D_0.Parameters.Path := 0; //Y then X
			MC_BR_MoveInPlane_Acp6D_0.Parameters.Mode := 0;
			MC_BR_MoveInPlane_Acp6D_0.Execute := TRUE;
			IF MC_BR_MoveInPlane_Acp6D_0.Acknowledge THEN
				MC_BR_MoveInPlane_Acp6D_0.Execute := FALSE;
				em.substate := 9004;
			END_IF

		9004:
			MC_BR_MoveInPlane_Acp6D_0.Parameters.Acceleration := gAcp6DCtrl.Par.Acceleration;
			MC_BR_MoveInPlane_Acp6D_0.Parameters.Velocity := gAcp6DCtrl.Par.Velocity;
			MC_BR_MoveInPlane_Acp6D_0.Shuttle := ADR(gAcp6DCtrl.Status.ShuttleInfo[4].shuttleRef);;
			MC_BR_MoveInPlane_Acp6D_0.Parameters.Position.X := gWorkstations[0].par.xLocation;;
			MC_BR_MoveInPlane_Acp6D_0.Parameters.Position.Y := gWorkstations[0].par.yLocation;
			MC_BR_MoveInPlane_Acp6D_0.Parameters.Path := 2; //Y then X
			MC_BR_MoveInPlane_Acp6D_0.Parameters.Mode := 0;
			MC_BR_MoveInPlane_Acp6D_0.Execute := TRUE;
			IF MC_BR_MoveInPlane_Acp6D_0.Acknowledge THEN
				MC_BR_MoveInPlane_Acp6D_0.Execute := FALSE;
				em.substate := 9005;
			END_IF

		9005:
			MC_BR_MoveInPlane_Acp6D_0.Parameters.Acceleration := gAcp6DCtrl.Par.Acceleration;
			MC_BR_MoveInPlane_Acp6D_0.Parameters.Velocity := gAcp6DCtrl.Par.Velocity;
			MC_BR_MoveInPlane_Acp6D_0.Shuttle := ADR(gAcp6DCtrl.Status.ShuttleInfo[5].shuttleRef);;
			MC_BR_MoveInPlane_Acp6D_0.Parameters.Position.X := gWorkstations[0].par.xLocation;;
			MC_BR_MoveInPlane_Acp6D_0.Parameters.Position.Y := gWorkstations[0].par.yLocation;
			MC_BR_MoveInPlane_Acp6D_0.Parameters.Path := 2; //Y then X
			MC_BR_MoveInPlane_Acp6D_0.Parameters.Mode := 0;
			MC_BR_MoveInPlane_Acp6D_0.Execute := TRUE;
			IF MC_BR_MoveInPlane_Acp6D_0.Acknowledge THEN
				MC_BR_MoveInPlane_Acp6D_0.Execute := FALSE;
				em.substate := 9006;
			END_IF

		9006:

	END_CASE

END_ACTION

ACTION conveyourStationMovement:
	// Setup
//	pWorkstation.MC_BR_MoveInPlane_Acp6D_0.Controller 					:= ADR(McAcp6DController);
//	pWorkstation.MC_BR_ShLevitation_Acp6D_0.Controller				:= ADR(McAcp6DController);
//	pWorkstation.MC_BR_MoveArcAngle_Acp6D_0.Controller					:= ADR(McAcp6DController);

	CASE cm.state OF
		// Display station at image
		//'<foreignObject x="20" y="20" width="300" height="300"><img src="Media/statusGreen.png" height="300" width="300"/>'
		//brsstrcat(ADR(showWorkStations),ADR('<foreingObject x="'));
		//brdkStrCat(ADR(showWorkStations), ADR(testDraw));
		//brdkStrCat(ADR(showWorkStations),'<foreingObject x="');

		0:
			//Check what shuttle is on top of workstation
			FOR k := 0 TO NUM_SHUTTLES DO
				IF((gAcp6DCtrl.Status.ShuttleInfo[k].Position.X > pWorkstation.par.xLocation - MARGIN AND gAcp6DCtrl.Status.ShuttleInfo[k].Position.X < pWorkstation.par.xLocation + MARGIN) AND
					gAcp6DCtrl.Status.ShuttleInfo[k].Position.Y > pWorkstation.par.yLocation - MARGIN AND gAcp6DCtrl.Status.ShuttleInfo[k].Position.Y < pWorkstation.par.yLocation + MARGIN) THEN
					IF gAcp6DCtrl.Status.ShuttleInfo[k].State = mcACP6D_SH_STATE_IDLING THEN
						pWorkstation.par.tempShuttleID := k;
						IF pWorkstation.par.landBeforeProcess THEN
							cm.state := 10;
						ELSE
							cm.state := 20;
						END_IF
					END_IF
				END_IF
			END_FOR

		10:
			//Land shuttle if reguired
			IF gAcp6DCtrl.Status.ShuttleInfo[pWorkstation.par.tempShuttleID].State = mcACP6D_SH_STATE_IDLING THEN
				pWorkstation.MC_BR_ShLevitation_Acp6D_0.Shuttle := ADR(gAcp6DCtrl.Status.ShuttleInfo[pWorkstation.par.tempShuttleID].shuttleRef);
				pWorkstation.MC_BR_ShLevitation_Acp6D_0.Parameters.Level := 0; //Land
				pWorkstation.MC_BR_ShLevitation_Acp6D_0.Parameters.Speed := 0;
				pWorkstation.MC_BR_ShLevitation_Acp6D_0.Execute := TRUE;
			END_IF
			IF pWorkstation.MC_BR_ShLevitation_Acp6D_0.Done THEN
				pWorkstation.MC_BR_ShLevitation_Acp6D_0.Execute := FALSE;
				cm.state := 20;
			END_IF

		20:
			//Simulate process TON timer
			pWorkstation.TON_0.PT := REAL_TO_TIME(pWorkstation.par.processTime*1000);
			pWorkstation.TON_0.IN := TRUE;
			IF pWorkstation.TON_0.Q THEN
				pWorkstation.TON_0.IN := FALSE;
				IF pWorkstation.par.landBeforeProcess THEN
					cm.state := 30;
				ELSE
					cm.state := 40;
				END_IF
			END_IF

		30:
			//Leviate shuttle if landed before process
			pWorkstation.MC_BR_ShLevitation_Acp6D_0.Shuttle := ADR(gAcp6DCtrl.Status.ShuttleInfo[pWorkstation.par.tempShuttleID].shuttleRef);
			pWorkstation.MC_BR_ShLevitation_Acp6D_0.Parameters.Level := 1; //Leviate
			pWorkstation.MC_BR_ShLevitation_Acp6D_0.Parameters.Speed := 0;
			pWorkstation.MC_BR_ShLevitation_Acp6D_0.Execute := TRUE;
			IF pWorkstation.MC_BR_ShLevitation_Acp6D_0.Done THEN
				pWorkstation.MC_BR_ShLevitation_Acp6D_0.Execute := FALSE;
				cm.state := 40;
			END_IF

		40:
			//Move to next workstation
			IF pWorkstation.par.ArcMovement THEN
				pWorkstation.MC_BR_MoveArc_Acp6D_0.Parameters.Angular.Center.X := 0.240;
				pWorkstation.MC_BR_MoveArc_Acp6D_0.Parameters.Angular.Center.Y := 0.240;
				pWorkstation.MC_BR_MoveArc_Acp6D_0.Parameters.Acceleration := gAcp6DCtrl.Par.Acceleration;
				pWorkstation.MC_BR_MoveArc_Acp6D_0.Parameters.Velocity := gAcp6DCtrl.Par.Velocity;
				pWorkstation.MC_BR_MoveArc_Acp6D_0.Parameters.Angular.Angle := 6.28318531; //360 degrees
				pWorkstation.MC_BR_MoveArc_Acp6D_0.Parameters.Mode := 0;
				pWorkstation.MC_BR_MoveArc_Acp6D_0.Shuttle := ADR(gAcp6DCtrl.Status.ShuttleInfo[pWorkstation.par.tempShuttleID].shuttleRef);
				pWorkstation.MC_BR_MoveArc_Acp6D_0.Execute := TRUE;
				IF pWorkstation.MC_BR_MoveArc_Acp6D_0.Acknowledge THEN
					pWorkstation.status.oneshot := FALSE;
					pWorkstation.MC_BR_MoveArc_Acp6D_0.Execute := FALSE;
					cm.state := 0;
				END_IF
			ELSE
				pWorkstation.MC_BR_MoveInPlane_Acp6D_0.Shuttle := ADR(gAcp6DCtrl.Status.ShuttleInfo[pWorkstation.par.tempShuttleID].shuttleRef);
				pWorkstation.MC_BR_MoveInPlane_Acp6D_0.Parameters.Velocity := gAcp6DCtrl.Par.Velocity;
				pWorkstation.MC_BR_MoveInPlane_Acp6D_0.Parameters.Acceleration := gAcp6DCtrl.Par.Acceleration;
				CASE i OF
					4:
						IF pWorkstation.workstationSwitcher THEN
							pWorkstation.MC_BR_MoveInPlane_Acp6D_0.Parameters.Position.X := gWorkstations[5].par.xLocation;
							pWorkstation.MC_BR_MoveInPlane_Acp6D_0.Parameters.Position.Y := gWorkstations[5].par.yLocation;
							pWorkstation.workstationSwitcher := FALSE;
						ELSE
							pWorkstation.MC_BR_MoveInPlane_Acp6D_0.Parameters.Position.X := gWorkstations[7].par.xLocation;
							pWorkstation.MC_BR_MoveInPlane_Acp6D_0.Parameters.Position.Y := gWorkstations[7].par.yLocation;
							pWorkstation.workstationSwitcher := TRUE;
						END_IF
					ELSE
						pWorkstation.MC_BR_MoveInPlane_Acp6D_0.Parameters.Position.X := gWorkstations[STRING_TO_UDINT(pWorkstation.par.nextStationSelector)].par.xLocation;
						pWorkstation.MC_BR_MoveInPlane_Acp6D_0.Parameters.Position.Y := gWorkstations[STRING_TO_UDINT(pWorkstation.par.nextStationSelector)].par.yLocation;
				END_CASE
				pWorkstation.MC_BR_MoveInPlane_Acp6D_0.Parameters.Mode := 0; //Absolute
				pWorkstation.MC_BR_MoveInPlane_Acp6D_0.Parameters.Path := pWorkstation.par.pathRouting; //0 Diagonal, 1 First X then Y, 2 First Y then X
				pWorkstation.MC_BR_MoveInPlane_Acp6D_0.Execute := TRUE;
				IF pWorkstation.MC_BR_MoveInPlane_Acp6D_0.Acknowledge THEN
					pWorkstation.status.oneshot := FALSE;
					pWorkstation.MC_BR_MoveInPlane_Acp6D_0.Execute := FALSE;
					cm.state := 0;
				END_IF
			END_IF
	END_CASE

	//Calls
	pWorkstation.MC_BR_MoveInPlane_Acp6D_0();
	pWorkstation.MC_BR_MoveArc_Acp6D_0();
	pWorkstation.MC_BR_ShLevitation_Acp6D_0();
	pWorkstation.TON_0();
	cm();

END_ACTION
```

#### workStationMovement.st
```iecst
ACTION workStationSetup:
	// Setup
	// Reset all workstations
	FOR i := 0 TO NR_OF_WORKSTATIONS DO
		gWorkstations[0].par.xLocation										:= 0.0;
		gWorkstations[0].par.yLocation										:= 0.0;
		gWorkstations[0].par.nextStationSelector							:= '0';
		gWorkstations[0].par.processTime									:= 0;
		gWorkstations[0].par.pathRouting									:= 0;
		gWorkstations[0].par.ArcMovement									:= FALSE;
		gWorkstations[0].par.landBeforeProcess								:= FALSE;
	END_FOR

	gWorkstations[0].par.xLocation										:= 0.180;
	gWorkstations[0].par.yLocation										:= 0.060;
	gWorkstations[0].par.nextStationSelector							:= '1';
	gWorkstations[0].par.processTime									:= 1;
	gWorkstations[0].par.pathRouting									:= 1;
	gWorkstations[0].par.ArcMovement									:= FALSE;
	gWorkstations[0].par.landBeforeProcess								:= FALSE;

	gWorkstations[1].par.xLocation										:= 0.540;
	gWorkstations[1].par.yLocation										:= 0.060;
	gWorkstations[1].par.nextStationSelector							:= '3';
	gWorkstations[1].par.processTime									:= 2;
	gWorkstations[1].par.pathRouting									:= 2;
	gWorkstations[1].par.ArcMovement									:= FALSE;
	gWorkstations[1].par.landBeforeProcess								:= FALSE;

	gWorkstations[2].par.xLocation										:= 0.660;
	gWorkstations[2].par.yLocation										:= 0.060;
	gWorkstations[2].par.nextStationSelector							:= '3';
	gWorkstations[2].par.processTime									:= 2;
	gWorkstations[2].par.pathRouting									:= 2;
	gWorkstations[2].par.ArcMovement									:= FALSE;
	gWorkstations[2].par.landBeforeProcess								:= FALSE;

	gWorkstations[3].par.xLocation										:= 0.660;
	gWorkstations[3].par.yLocation										:= 0.300;
	gWorkstations[3].par.nextStationSelector							:= '4';
	gWorkstations[3].par.processTime									:= 1;
	gWorkstations[3].par.pathRouting									:= 2;
	gWorkstations[3].par.ArcMovement									:= FALSE;
	gWorkstations[3].par.landBeforeProcess								:= FALSE;

	gWorkstations[4].par.xLocation										:= 0.540;
	gWorkstations[4].par.yLocation										:= 0.900;
	gWorkstations[4].par.nextStationSelector							:= '5';
	gWorkstations[4].par.processTime									:= 1;
	gWorkstations[4].par.pathRouting									:= 2;
	gWorkstations[4].par.ArcMovement									:= FALSE;
	gWorkstations[4].par.landBeforeProcess								:= FALSE;

	gWorkstations[5].par.xLocation										:= 0.540;
	gWorkstations[5].par.yLocation										:= 0.420;
	gWorkstations[5].par.nextStationSelector							:= '6';
	gWorkstations[5].par.processTime									:= 2;
	gWorkstations[5].par.pathRouting									:= 0;
	gWorkstations[5].par.ArcMovement									:= FALSE;
	gWorkstations[5].par.landBeforeProcess								:= FALSE;

	gWorkstations[6].par.xLocation										:= 0.060;
	gWorkstations[6].par.yLocation										:= 0.420;
	gWorkstations[6].par.nextStationSelector							:= '0';
	gWorkstations[6].par.processTime									:= 1;
	gWorkstations[6].par.pathRouting									:= 2;
	gWorkstations[6].par.ArcMovement									:= FALSE;
	gWorkstations[6].par.landBeforeProcess								:= FALSE;

	gWorkstations[7].par.xLocation										:= 0.300;
	gWorkstations[7].par.yLocation										:= 0.900;
	gWorkstations[7].par.nextStationSelector							:= '6';
	gWorkstations[7].par.processTime									:= 2;
	gWorkstations[7].par.pathRouting									:= 2;
	gWorkstations[7].par.ArcMovement									:= FALSE;
	gWorkstations[7].par.landBeforeProcess								:= FALSE;

	positionContainerWorkstationMov[0].initXPos							:= 0.060;
	positionContainerWorkstationMov[0].initYPos							:= 0.060;
	positionContainerWorkstationMov[1].initXPos							:= 0.180;
	positionContainerWorkstationMov[1].initYPos							:= 0.060;
	positionContainerWorkstationMov[2].initXPos							:= 0.420;
	positionContainerWorkstationMov[2].initYPos							:= 0.060;
	positionContainerWorkstationMov[3].initXPos							:= 0.540;
	positionContainerWorkstationMov[3].initYPos							:= 0.300;

	positionContainerWorkstationMov[4].initXPos							:= 0.060;
	positionContainerWorkstationMov[4].initYPos							:= 0.180;
	positionContainerWorkstationMov[5].initXPos							:= 0.060;
	positionContainerWorkstationMov[5].initYPos							:= 0.300;
	positionContainerWorkstationMov[6].initXPos							:= 0.660;
	positionContainerWorkstationMov[6].initYPos							:= 0.300;
	positionContainerWorkstationMov[7].initXPos							:= 0.540;
	positionContainerWorkstationMov[7].initYPos							:= 0.900;

	CASE em.substate OF
		8000:
			em.description := 'Move shuttle to pre pos';
			tempShuttleCounter := 0;
			MC_BR_MoveInPlaneAsync_Acp6D_0.Parameters.Acceleration := gAcp6DCtrl.Par.Acceleration;
			MC_BR_MoveInPlaneAsync_Acp6D_0.Parameters.Velocity := gAcp6DCtrl.Par.Velocity;
			FOR i := 0 TO UINT_TO_USINT(localCurrentNumShuttles-1) DO
				MC_BR_MoveInPlaneAsync_Acp6D_0.Parameters.AsyncPar[i].Shuttle := ADR(gAcp6DCtrl.Status.ShuttleInfo[i].shuttleRef);
				MC_BR_MoveInPlaneAsync_Acp6D_0.Parameters.AsyncPar[i].X := positionContainerWorkstationMov[i].initXPos;
				MC_BR_MoveInPlaneAsync_Acp6D_0.Parameters.AsyncPar[i].Y := positionContainerWorkstationMov[i].initYPos;
			END_FOR
			MC_BR_MoveInPlaneAsync_Acp6D_0.Execute := TRUE;
			IF MC_BR_MoveInPlaneAsync_Acp6D_0.Acknowledge THEN
				MC_BR_MoveInPlaneAsync_Acp6D_0.Execute := FALSE;
				em.substate := 8001;
			END_IF

		8001:
			MC_BR_MoveInPlane_Acp6D_0.Parameters.Acceleration := gAcp6DCtrl.Par.Acceleration;
			MC_BR_MoveInPlane_Acp6D_0.Parameters.Velocity := gAcp6DCtrl.Par.Velocity;
			MC_BR_MoveInPlane_Acp6D_0.Shuttle := ADR(gAcp6DCtrl.Status.ShuttleInfo[0].shuttleRef);;
			MC_BR_MoveInPlane_Acp6D_0.Parameters.Position.X := gWorkstations[0].par.xLocation;;
			MC_BR_MoveInPlane_Acp6D_0.Parameters.Position.Y := gWorkstations[0].par.yLocation;
			MC_BR_MoveInPlane_Acp6D_0.Parameters.Path := 0; //Y then X
			MC_BR_MoveInPlane_Acp6D_0.Parameters.Mode := 0;
			MC_BR_MoveInPlane_Acp6D_0.Execute := TRUE;
			IF MC_BR_MoveInPlane_Acp6D_0.Acknowledge THEN
				MC_BR_MoveInPlane_Acp6D_0.Execute := FALSE;
				em.substate := 8002;
			END_IF

		8002:
			MC_BR_MoveInPlane_Acp6D_0.Parameters.Acceleration := gAcp6DCtrl.Par.Acceleration;
			MC_BR_MoveInPlane_Acp6D_0.Parameters.Velocity := gAcp6DCtrl.Par.Velocity;
			MC_BR_MoveInPlane_Acp6D_0.Shuttle := ADR(gAcp6DCtrl.Status.ShuttleInfo[2].shuttleRef);;
			MC_BR_MoveInPlane_Acp6D_0.Parameters.Position.X := gWorkstations[1].par.xLocation;;
			MC_BR_MoveInPlane_Acp6D_0.Parameters.Position.Y := gWorkstations[1].par.yLocation;
			MC_BR_MoveInPlane_Acp6D_0.Parameters.Path := 0; //Y then X
			MC_BR_MoveInPlane_Acp6D_0.Parameters.Mode := 0;
			MC_BR_MoveInPlane_Acp6D_0.Execute := TRUE;
			IF MC_BR_MoveInPlane_Acp6D_0.Acknowledge THEN
				MC_BR_MoveInPlane_Acp6D_0.Execute := FALSE;
				em.substate := 8003;
			END_IF

		8003:
			MC_BR_MoveInPlane_Acp6D_0.Parameters.Acceleration := gAcp6DCtrl.Par.Acceleration;
			MC_BR_MoveInPlane_Acp6D_0.Parameters.Velocity := gAcp6DCtrl.Par.Velocity;
			MC_BR_MoveInPlane_Acp6D_0.Shuttle := ADR(gAcp6DCtrl.Status.ShuttleInfo[3].shuttleRef);;
			MC_BR_MoveInPlane_Acp6D_0.Parameters.Position.X := gWorkstations[3].par.xLocation;;
			MC_BR_MoveInPlane_Acp6D_0.Parameters.Position.Y := gWorkstations[3].par.yLocation;
			MC_BR_MoveInPlane_Acp6D_0.Parameters.Path := 0; //Y then X
			MC_BR_MoveInPlane_Acp6D_0.Parameters.Mode := 0;
			MC_BR_MoveInPlane_Acp6D_0.Execute := TRUE;
			IF MC_BR_MoveInPlane_Acp6D_0.Acknowledge THEN
				MC_BR_MoveInPlane_Acp6D_0.Execute := FALSE;
				em.substate := 8004;
			END_IF

		8004:
			MC_BR_MoveInPlane_Acp6D_0.Parameters.Acceleration := gAcp6DCtrl.Par.Acceleration;
			MC_BR_MoveInPlane_Acp6D_0.Parameters.Velocity := gAcp6DCtrl.Par.Velocity;
			MC_BR_MoveInPlane_Acp6D_0.Shuttle := ADR(gAcp6DCtrl.Status.ShuttleInfo[4].shuttleRef);;
			MC_BR_MoveInPlane_Acp6D_0.Parameters.Position.X := gWorkstations[0].par.xLocation;;
			MC_BR_MoveInPlane_Acp6D_0.Parameters.Position.Y := gWorkstations[0].par.yLocation;
			MC_BR_MoveInPlane_Acp6D_0.Parameters.Path := 2; //Y then X
			MC_BR_MoveInPlane_Acp6D_0.Parameters.Mode := 0;
			MC_BR_MoveInPlane_Acp6D_0.Execute := TRUE;
			IF MC_BR_MoveInPlane_Acp6D_0.Acknowledge THEN
				MC_BR_MoveInPlane_Acp6D_0.Execute := FALSE;
				em.substate := 8005;
			END_IF

		8005:
			MC_BR_MoveInPlane_Acp6D_0.Parameters.Acceleration := gAcp6DCtrl.Par.Acceleration;
			MC_BR_MoveInPlane_Acp6D_0.Parameters.Velocity := gAcp6DCtrl.Par.Velocity;
			MC_BR_MoveInPlane_Acp6D_0.Shuttle := ADR(gAcp6DCtrl.Status.ShuttleInfo[5].shuttleRef);;
			MC_BR_MoveInPlane_Acp6D_0.Parameters.Position.X := gWorkstations[0].par.xLocation;;
			MC_BR_MoveInPlane_Acp6D_0.Parameters.Position.Y := gWorkstations[0].par.yLocation;
			MC_BR_MoveInPlane_Acp6D_0.Parameters.Path := 2; //Y then X
			MC_BR_MoveInPlane_Acp6D_0.Parameters.Mode := 0;
			MC_BR_MoveInPlane_Acp6D_0.Execute := TRUE;
			IF MC_BR_MoveInPlane_Acp6D_0.Acknowledge THEN
				MC_BR_MoveInPlane_Acp6D_0.Execute := FALSE;
				em.substate := 8006;
			END_IF

		8006:

	END_CASE
END_ACTION

ACTION workStationMovement:

	CASE cm.state OF
		// Display station at image
		//'<foreignObject x="20" y="20" width="300" height="300"><img src="Media/statusGreen.png" height="300" width="300"/>'
		//brsstrcat(ADR(showWorkStations),ADR('<foreingObject x="'));
		//brdkStrCat(ADR(showWorkStations), ADR(testDraw));
		//brdkStrCat(ADR(showWorkStations),'<foreingObject x="');

		0:
			//Check what shuttle is on top of workstation
			FOR k := 0 TO NUM_SHUTTLES DO
				IF((gAcp6DCtrl.Status.ShuttleInfo[k].Position.X > pWorkstation.par.xLocation - MARGIN AND gAcp6DCtrl.Status.ShuttleInfo[k].Position.X < pWorkstation.par.xLocation + MARGIN) AND
					gAcp6DCtrl.Status.ShuttleInfo[k].Position.Y > pWorkstation.par.yLocation - MARGIN AND gAcp6DCtrl.Status.ShuttleInfo[k].Position.Y < pWorkstation.par.yLocation + MARGIN) THEN
					IF gAcp6DCtrl.Status.ShuttleInfo[k].State = mcACP6D_SH_STATE_IDLING THEN
						pWorkstation.par.tempShuttleID := k;
						IF pWorkstation.par.landBeforeProcess THEN
							cm.state := 10;
						ELSE
							cm.state := 20;
						END_IF
					END_IF
				END_IF
			END_FOR

		10:
			//Land shuttle if reguired
			IF gAcp6DCtrl.Status.ShuttleInfo[pWorkstation.par.tempShuttleID].State = mcACP6D_SH_STATE_IDLING THEN
				pWorkstation.MC_BR_ShLevitation_Acp6D_0.Shuttle := ADR(gAcp6DCtrl.Status.ShuttleInfo[pWorkstation.par.tempShuttleID].shuttleRef);
				pWorkstation.MC_BR_ShLevitation_Acp6D_0.Parameters.Level := 0; //Land
				pWorkstation.MC_BR_ShLevitation_Acp6D_0.Parameters.Speed := 10;
				pWorkstation.MC_BR_ShLevitation_Acp6D_0.Execute := TRUE;
			END_IF
			IF pWorkstation.MC_BR_ShLevitation_Acp6D_0.Done THEN
				pWorkstation.MC_BR_ShLevitation_Acp6D_0.Execute := FALSE;
				cm.state := 20;
			END_IF

		20:
			//Simulate process TON timer
			pWorkstation.TON_0.PT := REAL_TO_TIME(pWorkstation.par.processTime*1000);
			pWorkstation.TON_0.IN := TRUE;

			//Chooice which position shuttle stream to watch(Vision calc)
			CASE i OF
				3: shuttleToTakePictureOf := pWorkstation.par.tempShuttleID;
			END_CASE

			IF pWorkstation.TON_0.Q THEN
				pWorkstation.TON_0.IN := FALSE;
				IF pWorkstation.par.landBeforeProcess THEN
					cm.state := 30;
				ELSE
					cm.state := 40;
				END_IF
			END_IF

		30:
			//Leviate shuttle if landed before process
			pWorkstation.MC_BR_ShLevitation_Acp6D_0.Shuttle := ADR(gAcp6DCtrl.Status.ShuttleInfo[pWorkstation.par.tempShuttleID].shuttleRef);
			pWorkstation.MC_BR_ShLevitation_Acp6D_0.Parameters.Level := 1; //Leviate
			pWorkstation.MC_BR_ShLevitation_Acp6D_0.Parameters.Speed := 10;
			pWorkstation.MC_BR_ShLevitation_Acp6D_0.Execute := TRUE;
			IF pWorkstation.MC_BR_ShLevitation_Acp6D_0.Done THEN
				pWorkstation.MC_BR_ShLevitation_Acp6D_0.Execute := FALSE;
				cm.state := 40;
			END_IF

		40:
			//Move to next workstation
			pWorkstation.MC_BR_MoveInPlane_Acp6D_0.Shuttle := ADR(gAcp6DCtrl.Status.ShuttleInfo[pWorkstation.par.tempShuttleID].shuttleRef);
			pWorkstation.MC_BR_MoveInPlane_Acp6D_0.Parameters.Velocity := gAcp6DCtrl.Par.Velocity;
			pWorkstation.MC_BR_MoveInPlane_Acp6D_0.Parameters.Acceleration := gAcp6DCtrl.Par.Acceleration;
			pWorkstation.MC_BR_MoveInPlane_Acp6D_0.Parameters.Position.X := gWorkstations[STRING_TO_UDINT(pWorkstation.par.nextStationSelector)].par.xLocation;
			pWorkstation.MC_BR_MoveInPlane_Acp6D_0.Parameters.Position.Y := gWorkstations[STRING_TO_UDINT(pWorkstation.par.nextStationSelector)].par.yLocation;
			pWorkstation.MC_BR_MoveInPlane_Acp6D_0.Parameters.Mode := 0; //Absolute
			pWorkstation.MC_BR_MoveInPlane_Acp6D_0.Parameters.Path := pWorkstation.par.pathRouting; //0 Diagonal, 1 First X then Y, 2 First Y then X
			CASE i OF
				0:
					IF pWorkstation.workstationSwitcher AND NOT pWorkstation.status.oneshot THEN
						pWorkstation.MC_BR_MoveInPlane_Acp6D_0.Parameters.Position.X := gWorkstations[STRING_TO_UDINT(pWorkstation.par.nextStationSelector)].par.xLocation;
						pWorkstation.MC_BR_MoveInPlane_Acp6D_0.Parameters.Position.Y := gWorkstations[STRING_TO_UDINT(pWorkstation.par.nextStationSelector)].par.yLocation;
						pWorkstation.status.oneshot := TRUE;
						pWorkstation.workstationSwitcher := FALSE;
					ELSIF NOT pWorkstation.workstationSwitcher AND NOT pWorkstation.status.oneshot THEN
						pWorkstation.MC_BR_MoveInPlane_Acp6D_0.Parameters.Position.X := gWorkstations[STRING_TO_UDINT(pWorkstation.par.nextStationSelector)+1].par.xLocation;
						pWorkstation.MC_BR_MoveInPlane_Acp6D_0.Parameters.Position.Y := gWorkstations[STRING_TO_UDINT(pWorkstation.par.nextStationSelector)+1].par.yLocation;
						pWorkstation.status.oneshot := TRUE;
						pWorkstation.workstationSwitcher := TRUE;
					END_IF

				4:
					IF pWorkstation.workstationSwitcher THEN
						pWorkstation.MC_BR_MoveInPlane_Acp6D_0.Parameters.Position.X := gWorkstations[5].par.xLocation;
						pWorkstation.MC_BR_MoveInPlane_Acp6D_0.Parameters.Position.Y := gWorkstations[5].par.yLocation;
						pWorkstation.workstationSwitcher := FALSE;
					ELSE
						pWorkstation.MC_BR_MoveInPlane_Acp6D_0.Parameters.Position.X := gWorkstations[7].par.xLocation;
						pWorkstation.MC_BR_MoveInPlane_Acp6D_0.Parameters.Position.Y := gWorkstations[7].par.yLocation;
						pWorkstation.workstationSwitcher := TRUE;
					END_IF

			END_CASE
			pWorkstation.MC_BR_MoveInPlane_Acp6D_0.Execute := TRUE;
			IF pWorkstation.MC_BR_MoveInPlane_Acp6D_0.Acknowledge THEN
				pWorkstation.status.oneshot := FALSE;
				pWorkstation.MC_BR_MoveInPlane_Acp6D_0.Execute := FALSE;
				cm.state := 0;
			END_IF
	END_CASE

	//Calls
	pWorkstation.MC_BR_MoveInPlane_Acp6D_0();
	pWorkstation.MC_BR_ShLevitation_Acp6D_0();
	pWorkstation.TON_0();
	cm();

END_ACTION
```

#### flaskProgram.st
```iecst
ACTION flaskProgramTask:
	//setup
	positionContainerFlaskProgram[0].initXPos := 0.060;
	positionContainerFlaskProgram[0].initYPos := 0.060;
	positionContainerFlaskProgram[1].initXPos := 0.060;
	positionContainerFlaskProgram[1].initYPos := 0.180;
	positionContainerFlaskProgram[2].initXPos := 0.180;
	positionContainerFlaskProgram[2].initYPos := 0.120;
	positionContainerFlaskProgram[3].initXPos := 0.360;
	positionContainerFlaskProgram[3].initYPos := 0.120;
	positionContainerFlaskProgram[4].initXPos := 0.780;
	positionContainerFlaskProgram[4].initYPos := 0.900;
	positionContainerFlaskProgram[5].initXPos := 0.900;
	positionContainerFlaskProgram[5].initYPos := 0.900;
	positionContainerFlaskProgram[6].initXPos := 0.780;
	positionContainerFlaskProgram[6].initYPos := 0.780;
	positionContainerFlaskProgram[7].initXPos := 0.900;
	positionContainerFlaskProgram[7].initYPos := 0.780;
	positionContainerFlaskProgram[8].initXPos := 0.780;
	positionContainerFlaskProgram[8].initYPos := 0.660;
	positionContainerFlaskProgram[9].initXPos := 0.900;
	positionContainerFlaskProgram[9].initYPos := 0.660;
	CASE em.substate OF
		12000:
			em.description := 'Move shuttle to pre pos';
			tempShuttleCounter := 0;
			MC_BR_MoveInPlaneAsync_Acp6D_0.Parameters.Acceleration := gAcp6DCtrl.Par.Acceleration;
			MC_BR_MoveInPlaneAsync_Acp6D_0.Parameters.Velocity := gAcp6DCtrl.Par.Velocity;
			FOR i := 0 TO UINT_TO_USINT(localCurrentNumShuttles-1) DO
				MC_BR_MoveInPlaneAsync_Acp6D_0.Parameters.AsyncPar[i].Shuttle := ADR(gAcp6DCtrl.Status.ShuttleInfo[i].shuttleRef);
				MC_BR_MoveInPlaneAsync_Acp6D_0.Parameters.AsyncPar[i].X := positionContainerFlaskProgram[i].initXPos;
				MC_BR_MoveInPlaneAsync_Acp6D_0.Parameters.AsyncPar[i].Y := positionContainerFlaskProgram[i].initYPos;
			END_FOR
			MC_BR_MoveInPlaneAsync_Acp6D_0.Execute := TRUE;
			IF MC_BR_MoveInPlaneAsync_Acp6D_0.Done THEN
				MC_BR_MoveInPlaneAsync_Acp6D_0.Execute := FALSE;
				em.substate := 12010;
			END_IF

		12010:
			em.description := 'Start circle movement on shuttle 4';
			MC_BR_MoveArc_Acp6D_0.Shuttle := ADR(gAcp6DCtrl.Status.ShuttleInfo[3].shuttleRef);
			MC_BR_MoveArc_Acp6D_0.Parameters.Option := mcACP6D_ARC_ANGULAR;
			MC_BR_MoveArc_Acp6D_0.Parameters.Acceleration := flaskProgramAcceleration;
			MC_BR_MoveArc_Acp6D_0.Parameters.Velocity := flaskProgramVelocity;
			MC_BR_MoveArc_Acp6D_0.Parameters.Angular.Center.X := 0.361;
			MC_BR_MoveArc_Acp6D_0.Parameters.Angular.Center.Y := 0.120;
			MC_BR_MoveArc_Acp6D_0.Parameters.Angular.Angle := 6283.1;
			MC_BR_MoveArc_Acp6D_0.Parameters.Mode := 0; //Abs
			MC_BR_MoveArc_Acp6D_0.Parameters.Direction := 0; //Clockwise
			MC_BR_MoveArc_Acp6D_0.Execute := TRUE;
			IF MC_BR_MoveArc_Acp6D_0.Acknowledge THEN
				MC_BR_MoveArc_Acp6D_0.Execute := FALSE;
				em.substate := 12020;
			END_IF

		12020:
			em.description := 'shuttle 1,2,3 is doing basic movement, shuttle 4 is rotation from command above';

	END_CASE

END_ACTION
```

#### boxProgram.st
```iecst
ACTION boxProgramTask:

//	positionContainerBoxProgram[0].initXPos := 0.060;
//	positionContainerBoxProgram[0].initYPos := 0.180;
//	positionContainerBoxProgram[1].initXPos := 0.180;
//	positionContainerBoxProgram[1].initYPos := 0.060;
//	positionContainerBoxProgram[2].initXPos := 0.420;
//	positionContainerBoxProgram[2].initYPos := 0.180;
//	positionContainerBoxProgram[3].initXPos := 0.420;
//	positionContainerBoxProgram[3].initYPos := 0.060;

	CASE em.substate OF
		13000:
			em.description := 'Move shuttle to pre pos';
			positionContainerBoxProgram[0].initXPos := 0.060;
			positionContainerBoxProgram[0].initYPos := 0.180;
			positionContainerBoxProgram[1].initXPos := 0.180;
			positionContainerBoxProgram[1].initYPos := 0.060;
			positionContainerBoxProgram[2].initXPos := 0.540;
			positionContainerBoxProgram[2].initYPos := 0.540;
			positionContainerBoxProgram[3].initXPos := 0.660;
			positionContainerBoxProgram[3].initYPos := 0.540;

			positionContainerBoxProgram[4].initXPos := 0.540;
			positionContainerBoxProgram[4].initYPos := 0.900;
			positionContainerBoxProgram[5].initXPos := 0.660;
			positionContainerBoxProgram[5].initYPos := 0.900;
			positionContainerBoxProgram[6].initXPos := 0.540;
			positionContainerBoxProgram[6].initYPos := 0.780;
			positionContainerBoxProgram[7].initXPos := 0.660;
			positionContainerBoxProgram[7].initYPos := 0.780;

			tempShuttleCounter := 0;
			MC_BR_MoveInPlaneAsync_Acp6D_0.Parameters.Acceleration := gAcp6DCtrl.Par.Acceleration;
			MC_BR_MoveInPlaneAsync_Acp6D_0.Parameters.Velocity := gAcp6DCtrl.Par.Velocity;
			FOR i := 0 TO UINT_TO_USINT(localCurrentNumShuttles-1) DO
				MC_BR_MoveInPlaneAsync_Acp6D_0.Parameters.AsyncPar[i].Shuttle := ADR(gAcp6DCtrl.Status.ShuttleInfo[i].shuttleRef);
				MC_BR_MoveInPlaneAsync_Acp6D_0.Parameters.AsyncPar[i].X := positionContainerBoxProgram[i].initXPos;
				MC_BR_MoveInPlaneAsync_Acp6D_0.Parameters.AsyncPar[i].Y := positionContainerBoxProgram[i].initYPos;
			END_FOR
			MC_BR_MoveInPlaneAsync_Acp6D_0.Execute := TRUE;
			IF MC_BR_MoveInPlaneAsync_Acp6D_0.Acknowledge THEN
				cmdBoxProgram.LastTypeWasBox := TRUE;
				MC_BR_MoveInPlaneAsync_Acp6D_0.Execute := FALSE;
				em.substate := 13010;
			END_IF

		13010:
			em.description := 'Select size or start from HMI';
			IF cmdBoxProgram.smallBox OR cmdBoxProgram.bigBox THEN
				IF cmdBoxProgram.LastTypeWasBox THEN
					em.substate := 13020;
				ELSE
					em.substate := 13015;
				END_IF
			ELSIF cmdBoxProgram.bottle THEN
				IF cmdBoxProgram.LastTypeWasBox THEN
					em.substate := 13011;
				ELSE
					em.substate := 13030;
				END_IF
			END_IF

		13011:
			em.description := 'move shuttle away';
			MC_BR_MoveInPlane_Acp6D_0.Shuttle := ADR(gAcp6DCtrl.Status.ShuttleInfo[0].shuttleRef);
			MC_BR_MoveInPlane_Acp6D_0.Parameters.Position.X := 0.300; // at 0.180 = 80mm on x box
			MC_BR_MoveInPlane_Acp6D_0.Parameters.Position.Y := 0.300; // at 0.060 = 80mm on y box
			MC_BR_MoveInPlane_Acp6D_0.Parameters.Velocity := gAcp6DCtrl.Par.Velocity;
			MC_BR_MoveInPlane_Acp6D_0.Parameters.Acceleration := gAcp6DCtrl.Par.Acceleration;
			MC_BR_MoveInPlane_Acp6D_0.Parameters.Mode := 0;
			MC_BR_MoveInPlane_Acp6D_0.Parameters.Path := 2; //Y then X
			MC_BR_MoveInPlane_Acp6D_0.Execute := TRUE;
			IF MC_BR_MoveInPlane_Acp6D_0.Done THEN
				MC_BR_MoveInPlane_Acp6D_0.Execute := FALSE;
				em.substate := 13012;
			END_IF

		13012:
			em.description := 'move shuttle 1 to correct pos';
			MC_BR_MoveInPlane_Acp6D_0.Shuttle := ADR(gAcp6DCtrl.Status.ShuttleInfo[1].shuttleRef);
			MC_BR_MoveInPlane_Acp6D_0.Parameters.Position.X := 0.060; // at 0.180 = 80mm on x box
			MC_BR_MoveInPlane_Acp6D_0.Parameters.Position.Y := 0.060; // at 0.060 = 80mm on y box
			MC_BR_MoveInPlane_Acp6D_0.Parameters.Velocity := gAcp6DCtrl.Par.Velocity;
			MC_BR_MoveInPlane_Acp6D_0.Parameters.Acceleration := gAcp6DCtrl.Par.Acceleration;
			MC_BR_MoveInPlane_Acp6D_0.Parameters.Mode := 0;
			MC_BR_MoveInPlane_Acp6D_0.Parameters.Path := 0; //X then Y
			MC_BR_MoveInPlane_Acp6D_0.Execute := TRUE;
			IF MC_BR_MoveInPlane_Acp6D_0.Done THEN
				MC_BR_MoveInPlane_Acp6D_0.Execute := FALSE;
				cmdBoxProgram.LastTypeWasBox := FALSE;
				em.substate := 13010;
			END_IF

		13015:
			em.description := 'adjust shuttle to box';
			MC_BR_MoveInPlane_Acp6D_0.Shuttle := ADR(gAcp6DCtrl.Status.ShuttleInfo[1].shuttleRef);
			MC_BR_MoveInPlane_Acp6D_0.Parameters.Position.X := 0.300; // at 0.180 = 80mm on x box
			MC_BR_MoveInPlane_Acp6D_0.Parameters.Position.Y := 0.060; // at 0.060 = 80mm on y box
			MC_BR_MoveInPlane_Acp6D_0.Parameters.Velocity := gAcp6DCtrl.Par.Velocity;
			MC_BR_MoveInPlane_Acp6D_0.Parameters.Acceleration := gAcp6DCtrl.Par.Acceleration;
			MC_BR_MoveInPlane_Acp6D_0.Parameters.Mode := 0;
			MC_BR_MoveInPlane_Acp6D_0.Parameters.Path := 0; //Y then X
			MC_BR_MoveInPlane_Acp6D_0.Execute := TRUE;
			IF MC_BR_MoveInPlane_Acp6D_0.Done THEN
				MC_BR_MoveInPlane_Acp6D_0.Execute := FALSE;
				em.substate := 13016;
			END_IF

		13016:
			em.description := 'adjust shuttle to box';
			MC_BR_MoveInPlane_Acp6D_0.Shuttle := ADR(gAcp6DCtrl.Status.ShuttleInfo[0].shuttleRef);
			MC_BR_MoveInPlane_Acp6D_0.Parameters.Position.X := 0.060; // at 0.180 = 80mm on x box
			MC_BR_MoveInPlane_Acp6D_0.Parameters.Position.Y := 0.180; // at 0.060 = 80mm on y box
			MC_BR_MoveInPlane_Acp6D_0.Parameters.Velocity := gAcp6DCtrl.Par.Velocity;
			MC_BR_MoveInPlane_Acp6D_0.Parameters.Acceleration := gAcp6DCtrl.Par.Acceleration;
			MC_BR_MoveInPlane_Acp6D_0.Parameters.Mode := 0;
			MC_BR_MoveInPlane_Acp6D_0.Parameters.Path := 0; //Y then X
			MC_BR_MoveInPlane_Acp6D_0.Execute := TRUE;
			IF MC_BR_MoveInPlane_Acp6D_0.Done THEN
				MC_BR_MoveInPlane_Acp6D_0.Execute := FALSE;
				cmdBoxProgram.LastTypeWasBox := TRUE;
				em.substate := 13010;
			END_IF

		13020:
			IF cmdBoxProgram.smallBox THEN
				cmdBoxProgram.smallBox := FALSE;
				em.substate := 13100;
			ELSIF cmdBoxProgram.bigBox THEN
				cmdBoxProgram.bigBox := FALSE;
				em.substate := 13200;
			END_IF

		13030:
			em.description := 'which bottle?';
			IF cmdBoxProgram.bottle THEN
				cmdBoxProgram.bottle := FALSE;
				em.substate := 13250;
			END_IF

		13100:
			em.description := 'adjust shuttle to small size box';
			MC_BR_MoveInPlane_Acp6D_0.Shuttle := ADR(gAcp6DCtrl.Status.ShuttleInfo[1].shuttleRef);
			MC_BR_MoveInPlane_Acp6D_0.Parameters.Position.X := 0.2175; // at 0.180 = 80mm on x box
			MC_BR_MoveInPlane_Acp6D_0.Parameters.Position.Y := 0.084; // at 0.060 = 80mm on y box
			MC_BR_MoveInPlane_Acp6D_0.Parameters.Velocity := gAcp6DCtrl.Par.Velocity;
			MC_BR_MoveInPlane_Acp6D_0.Parameters.Acceleration := gAcp6DCtrl.Par.Acceleration;
			MC_BR_MoveInPlane_Acp6D_0.Parameters.Mode := 0;
			MC_BR_MoveInPlane_Acp6D_0.Parameters.Path := 0; //Y then X
			MC_BR_MoveInPlane_Acp6D_0.Execute := TRUE;
			IF MC_BR_MoveInPlane_Acp6D_0.Acknowledge THEN
				MC_BR_MoveInPlane_Acp6D_0.Execute := FALSE;
				em.substate := 13300;
			END_IF

		13200:
			em.description := 'adjust shuttle to big size box';
			MC_BR_MoveInPlane_Acp6D_0.Shuttle := ADR(gAcp6DCtrl.Status.ShuttleInfo[1].shuttleRef);
			MC_BR_MoveInPlane_Acp6D_0.Parameters.Position.X := 0.229; // at 0.180 = 80mm on x box
			MC_BR_MoveInPlane_Acp6D_0.Parameters.Position.Y := 0.066; // at 0.060 = 80mm on y box
			MC_BR_MoveInPlane_Acp6D_0.Parameters.Velocity := gAcp6DCtrl.Par.Velocity;
			MC_BR_MoveInPlane_Acp6D_0.Parameters.Acceleration := gAcp6DCtrl.Par.Acceleration;
			MC_BR_MoveInPlane_Acp6D_0.Parameters.Mode := 0;
			MC_BR_MoveInPlane_Acp6D_0.Parameters.Path := 0; //Y then X
			MC_BR_MoveInPlane_Acp6D_0.Execute := TRUE;
			IF MC_BR_MoveInPlane_Acp6D_0.Acknowledge THEN
				MC_BR_MoveInPlane_Acp6D_0.Execute := FALSE;
				em.substate := 13300;
			END_IF

		13250:
			em.description := 'adjust shuttle to bottle';
			MC_BR_MoveInPlane_Acp6D_0.Shuttle := ADR(gAcp6DCtrl.Status.ShuttleInfo[0].shuttleRef);
			MC_BR_MoveInPlane_Acp6D_0.Parameters.Position.X := 0.132; // at 0.180 = 80mm on x box
			MC_BR_MoveInPlane_Acp6D_0.Parameters.Position.Y := 0.181; // at 0.060 = 80mm on y box
			MC_BR_MoveInPlane_Acp6D_0.Parameters.Velocity := gAcp6DCtrl.Par.Velocity;
			MC_BR_MoveInPlane_Acp6D_0.Parameters.Acceleration := gAcp6DCtrl.Par.Acceleration;
			MC_BR_MoveInPlane_Acp6D_0.Parameters.Mode := 0;
			MC_BR_MoveInPlane_Acp6D_0.Parameters.Path := 0; //Y then X
			MC_BR_MoveInPlane_Acp6D_0.Execute := TRUE;
			IF MC_BR_MoveInPlane_Acp6D_0.Acknowledge THEN
				MC_BR_MoveInPlane_Acp6D_0.Execute := FALSE;
				em.substate := 13310;
			END_IF

		13300:
			em.description := 'start timer';
			TON_0.PT := t#3s;
			TON_0.IN := TRUE;
			IF TON_0.Q THEN
				TON_0.IN := FALSE;
				em.substate := 13330;
			END_IF

		13310:
			em.description := 'start timer';
			TON_0.PT := t#3s;
			TON_0.IN := TRUE;
			IF TON_0.Q THEN
				TON_0.IN := FALSE;
				em.substate := 13500;
			END_IF

		13330:
			em.description := 'Couple ShuttleGroup1_2';
			MC_BR_ShGroupCoupleCtrl_Acp6D_0.ShuttleGroup := shGroupShuttle1_2;
			MC_BR_ShGroupCoupleCtrl_Acp6D_0.Parameters.Mode := 1;
			MC_BR_ShGroupCoupleCtrl_Acp6D_0.Parameters.Option := 1; //Couple
			MC_BR_ShGroupCoupleCtrl_Acp6D_0.Execute := TRUE;
			IF MC_BR_ShGroupCoupleCtrl_Acp6D_0.Done THEN
				MC_BR_ShGroupCoupleCtrl_Acp6D_0.Execute := FALSE;
				em.substate := 13340;
			END_IF

		13340:
			em.description := 'Move box around';
			MC_BR_MoveInPlane_Acp6D_0.Shuttle := ADR(gAcp6DCtrl.Status.ShuttleInfo[0].shuttleRef);;
			MC_BR_MoveInPlane_Acp6D_0.Parameters.Position.X := 0.500;
			MC_BR_MoveInPlane_Acp6D_0.Parameters.Position.Y := 0.420;
			MC_BR_MoveInPlane_Acp6D_0.Parameters.Velocity := 1;
			MC_BR_MoveInPlane_Acp6D_0.Parameters.Acceleration := 1;
			MC_BR_MoveInPlane_Acp6D_0.Parameters.Path := 2; //Y then X
			MC_BR_MoveInPlane_Acp6D_0.Parameters.Mode := 0;
			MC_BR_MoveInPlane_Acp6D_0.Execute := TRUE;
			IF MC_BR_MoveInPlane_Acp6D_0.Acknowledge THEN
				MC_BR_MoveInPlane_Acp6D_0.Execute := FALSE;
				em.substate := 13360;
			END_IF

		13360:
			MC_BR_MoveInPlane_Acp6D_0.Shuttle := ADR(gAcp6DCtrl.Status.ShuttleInfo[0].shuttleRef);;
			MC_BR_MoveInPlane_Acp6D_0.Parameters.Position.X := 0.060;
			MC_BR_MoveInPlane_Acp6D_0.Parameters.Position.Y := 0.180;
			MC_BR_MoveInPlane_Acp6D_0.Parameters.Velocity := 1;
			MC_BR_MoveInPlane_Acp6D_0.Parameters.Acceleration := 1;
			MC_BR_MoveInPlane_Acp6D_0.Parameters.Path := 2;
			MC_BR_MoveInPlane_Acp6D_0.Parameters.Mode := 0;
			MC_BR_MoveInPlane_Acp6D_0.Execute := TRUE;
			IF MC_BR_MoveInPlane_Acp6D_0.Acknowledge THEN
				MC_BR_MoveInPlane_Acp6D_0.Execute := FALSE;
				em.substate := 13400;
			END_IF

//		13350:
//			em.description := 'Move shuttles in X Y and RZ at the same time';
//			MC_BR_Move6D_Acp6D_0.Parameters.InPlane.Acceleration := 0.5;
//			MC_BR_Move6D_Acp6D_0.Parameters.InPlane.Velocity := 0.14;
//			MC_BR_Move6D_Acp6D_0.Shuttle := ADR(gAcp6DCtrl.Status.ShuttleInfo[0].shuttleRef);
//			MC_BR_Move6D_Acp6D_0.Parameters.ShortAxis.Velocity.Rz := MC_BR_Move6D_Acp6D_0.Parameters.ShortAxis.Velocity.Ry := MC_BR_Move6D_Acp6D_0.Parameters.ShortAxis.Velocity.Rx := MC_BR_Move6D_Acp6D_0.Parameters.ShortAxis.Velocity.Z := 0.300;
//			MC_BR_Move6D_Acp6D_0.Parameters.InPlane.Position.X := 0.125;
//			MC_BR_Move6D_Acp6D_0.Parameters.InPlane.Position.Y := 0.180;
//			MC_BR_Move6D_Acp6D_0.Parameters.ShortAxis.Position.Z := 0.001;
//			MC_BR_Move6D_Acp6D_0.Parameters.ShortAxis.Position.Rx := 0;
//			MC_BR_Move6D_Acp6D_0.Parameters.ShortAxis.Position.Ry := 0;
//			MC_BR_Move6D_Acp6D_0.Parameters.ShortAxis.Position.Rz := 0.125;
//			MC_BR_Move6D_Acp6D_0.Execute := TRUE;
//			IF MC_BR_Move6D_Acp6D_0.Acknowledge THEN
//				MC_BR_Move6D_Acp6D_0.Execute := FALSE;
//				em.substate := 13360;
//			END_IF
//
//		13360:
//			em.description := 'Move shuttles in X Y and RZ at the same time';
//			MC_BR_Move6D_Acp6D_0.Parameters.InPlane.Acceleration := 0.5;
//			MC_BR_Move6D_Acp6D_0.Parameters.InPlane.Velocity := 0.14;
//			MC_BR_Move6D_Acp6D_0.Shuttle := ADR(gAcp6DCtrl.Status.ShuttleInfo[0].shuttleRef);
//			MC_BR_Move6D_Acp6D_0.Parameters.ShortAxis.Velocity.Rz := MC_BR_Move6D_Acp6D_0.Parameters.ShortAxis.Velocity.Ry := MC_BR_Move6D_Acp6D_0.Parameters.ShortAxis.Velocity.Rx := MC_BR_Move6D_Acp6D_0.Parameters.ShortAxis.Velocity.Z := 0.300;
//			MC_BR_Move6D_Acp6D_0.Parameters.InPlane.Position.X := 0.125;
//			MC_BR_Move6D_Acp6D_0.Parameters.InPlane.Position.Y := 0.180;
//			MC_BR_Move6D_Acp6D_0.Parameters.ShortAxis.Position.Z := 0.001;
//			MC_BR_Move6D_Acp6D_0.Parameters.ShortAxis.Position.Rx := 0;
//			MC_BR_Move6D_Acp6D_0.Parameters.ShortAxis.Position.Ry := 0;
//			MC_BR_Move6D_Acp6D_0.Parameters.ShortAxis.Position.Rz := -0.125;
//			MC_BR_Move6D_Acp6D_0.Execute := TRUE;
//			IF MC_BR_Move6D_Acp6D_0.Acknowledge THEN
//				MC_BR_Move6D_Acp6D_0.Execute := FALSE;
//				em.substate := 13370;
//			END_IF
//
//		13370:
//			em.description := 'Move shuttles in X Y and RZ at the same time';
//			MC_BR_Move6D_Acp6D_0.Parameters.InPlane.Acceleration := 0.5;
//			MC_BR_Move6D_Acp6D_0.Parameters.InPlane.Velocity := 0.14;
//			MC_BR_Move6D_Acp6D_0.Shuttle := ADR(gAcp6DCtrl.Status.ShuttleInfo[0].shuttleRef);
//			MC_BR_Move6D_Acp6D_0.Parameters.ShortAxis.Velocity.Rz := MC_BR_Move6D_Acp6D_0.Parameters.ShortAxis.Velocity.Ry := MC_BR_Move6D_Acp6D_0.Parameters.ShortAxis.Velocity.Rx := MC_BR_Move6D_Acp6D_0.Parameters.ShortAxis.Velocity.Z := 0.300;
//			MC_BR_Move6D_Acp6D_0.Parameters.InPlane.Position.X := 0.060;
//			MC_BR_Move6D_Acp6D_0.Parameters.InPlane.Position.Y := 0.180;
//			MC_BR_Move6D_Acp6D_0.Parameters.ShortAxis.Position.Z := 0.001;
//			MC_BR_Move6D_Acp6D_0.Parameters.ShortAxis.Position.Rx := 0;
//			MC_BR_Move6D_Acp6D_0.Parameters.ShortAxis.Position.Ry := 0;
//			MC_BR_Move6D_Acp6D_0.Parameters.ShortAxis.Position.Rz := 0.125;
//			MC_BR_Move6D_Acp6D_0.Execute := TRUE;
//			IF MC_BR_Move6D_Acp6D_0.Acknowledge THEN
//				MC_BR_Move6D_Acp6D_0.Execute := FALSE;
//				em.substate := 13380;
//			END_IF
//
//		13380:
//			em.description := 'Move shuttles in X Y and RZ at the same time';
//			MC_BR_Move6D_Acp6D_0.Parameters.InPlane.Acceleration := 0.5;
//			MC_BR_Move6D_Acp6D_0.Parameters.InPlane.Velocity := 0.14;
//			MC_BR_Move6D_Acp6D_0.Shuttle := ADR(gAcp6DCtrl.Status.ShuttleInfo[0].shuttleRef);
//			MC_BR_Move6D_Acp6D_0.Parameters.ShortAxis.Velocity.Rz := MC_BR_Move6D_Acp6D_0.Parameters.ShortAxis.Velocity.Ry := MC_BR_Move6D_Acp6D_0.Parameters.ShortAxis.Velocity.Rx := MC_BR_Move6D_Acp6D_0.Parameters.ShortAxis.Velocity.Z := 0.300;
//			MC_BR_Move6D_Acp6D_0.Parameters.InPlane.Position.X := 0.125;
//			MC_BR_Move6D_Acp6D_0.Parameters.InPlane.Position.Y := 0.180;
//			MC_BR_Move6D_Acp6D_0.Parameters.ShortAxis.Position.Z := 0.001;
//			MC_BR_Move6D_Acp6D_0.Parameters.ShortAxis.Position.Rx := 0;
//			MC_BR_Move6D_Acp6D_0.Parameters.ShortAxis.Position.Ry := 0;
//			MC_BR_Move6D_Acp6D_0.Parameters.ShortAxis.Position.Rz := -0.125;
//			MC_BR_Move6D_Acp6D_0.Execute := TRUE;
//			IF MC_BR_Move6D_Acp6D_0.Acknowledge THEN
//				MC_BR_Move6D_Acp6D_0.Execute := FALSE;
//				em.substate := 13390;
//			END_IF
//
//		13390:
//			em.description := 'Move shuttles in X Y and RZ at the same time';
//			MC_BR_Move6D_Acp6D_0.Parameters.InPlane.Acceleration := 0.5;
//			MC_BR_Move6D_Acp6D_0.Parameters.InPlane.Velocity := 0.14;
//			MC_BR_Move6D_Acp6D_0.Shuttle := ADR(gAcp6DCtrl.Status.ShuttleInfo[0].shuttleRef);
//			MC_BR_Move6D_Acp6D_0.Parameters.ShortAxis.Velocity.Rz := MC_BR_Move6D_Acp6D_0.Parameters.ShortAxis.Velocity.Ry := MC_BR_Move6D_Acp6D_0.Parameters.ShortAxis.Velocity.Rx := MC_BR_Move6D_Acp6D_0.Parameters.ShortAxis.Velocity.Z := 0.300;
//			MC_BR_Move6D_Acp6D_0.Parameters.InPlane.Position.X := 0.060;
//			MC_BR_Move6D_Acp6D_0.Parameters.InPlane.Position.Y := 0.180;
//			MC_BR_Move6D_Acp6D_0.Parameters.ShortAxis.Position.Z := 0.001;
//			MC_BR_Move6D_Acp6D_0.Parameters.ShortAxis.Position.Rx := 0;
//			MC_BR_Move6D_Acp6D_0.Parameters.ShortAxis.Position.Ry := 0;
//			MC_BR_Move6D_Acp6D_0.Parameters.ShortAxis.Position.Rz := 0;
//			MC_BR_Move6D_Acp6D_0.Execute := TRUE;
//			IF MC_BR_Move6D_Acp6D_0.Acknowledge THEN
//				MC_BR_Move6D_Acp6D_0.Execute := FALSE;
//				em.substate := 13400;
//			END_IF

		13400:
			em.description := 'DeCouple ShuttleGroup1_2';
			MC_BR_ShGroupCoupleCtrl_Acp6D_0.ShuttleGroup := shGroupShuttle1_2;
			MC_BR_ShGroupCoupleCtrl_Acp6D_0.Parameters.Option := 0; //DeCouple
			MC_BR_ShGroupCoupleCtrl_Acp6D_0.Execute := TRUE;
			IF MC_BR_ShGroupCoupleCtrl_Acp6D_0.Done THEN
				MC_BR_ShGroupCoupleCtrl_Acp6D_0.Execute := FALSE;
				em.substate := 13010;
			END_IF

		13500:
			em.description := 'Couple ShuttleGroup1_2';
			MC_BR_ShGroupCoupleCtrl_Acp6D_0.ShuttleGroup := shGroupShuttle1_2;
			MC_BR_ShGroupCoupleCtrl_Acp6D_0.Parameters.Mode := 1;
			MC_BR_ShGroupCoupleCtrl_Acp6D_0.Parameters.Option := 1; //Couple
			MC_BR_ShGroupCoupleCtrl_Acp6D_0.Execute := TRUE;
			IF MC_BR_ShGroupCoupleCtrl_Acp6D_0.Done THEN
				MC_BR_ShGroupCoupleCtrl_Acp6D_0.Execute := FALSE;
				em.substate := 13510;
			END_IF

		13510:
			em.description := 'Move bottle around';
			MC_BR_MoveInPlane_Acp6D_0.Shuttle := ADR(gAcp6DCtrl.Status.ShuttleInfo[1].shuttleRef);;
			MC_BR_MoveInPlane_Acp6D_0.Parameters.Position.X := 0.540;
			MC_BR_MoveInPlane_Acp6D_0.Parameters.Position.Y := 0.290;
			MC_BR_MoveInPlane_Acp6D_0.Parameters.Velocity := 1;
			MC_BR_MoveInPlane_Acp6D_0.Parameters.Acceleration := 1;
			MC_BR_MoveInPlane_Acp6D_0.Parameters.Path := 2; //Y then X
			MC_BR_MoveInPlane_Acp6D_0.Parameters.Mode := 0;
			MC_BR_MoveInPlane_Acp6D_0.Execute := TRUE;
			IF MC_BR_MoveInPlane_Acp6D_0.Acknowledge THEN
				MC_BR_MoveInPlane_Acp6D_0.Execute := FALSE;
				em.substate := 13530;
			END_IF

		13530:
			em.description := 'Move bottle around';
			MC_BR_MoveInPlane_Acp6D_0.Shuttle := ADR(gAcp6DCtrl.Status.ShuttleInfo[1].shuttleRef);;
			MC_BR_MoveInPlane_Acp6D_0.Parameters.Position.X := 0.060;
			MC_BR_MoveInPlane_Acp6D_0.Parameters.Position.Y := 0.060;
			MC_BR_MoveInPlane_Acp6D_0.Parameters.Velocity := 1;
			MC_BR_MoveInPlane_Acp6D_0.Parameters.Acceleration := 1;
			MC_BR_MoveInPlane_Acp6D_0.Parameters.Path := 2;
			MC_BR_MoveInPlane_Acp6D_0.Parameters.Mode := 0;
			MC_BR_MoveInPlane_Acp6D_0.Execute := TRUE;
			IF MC_BR_MoveInPlane_Acp6D_0.Acknowledge THEN
				MC_BR_MoveInPlane_Acp6D_0.Execute := FALSE;
				em.substate := 13400; //decouple state
			END_IF
	END_CASE

	TON_0();

END_ACTION
```
